C05488=1193.107,194.076,-58.104,-177.783,6.528,148.541
C05489=1193.102,194.324,-58.128,-177.781,6.530,148.540
C05490=1193.099,194.573,-58.150,-177.778,6.532,148.540
C05491=1193.094,194.822,-58.174,-177.775,6.534,148.540
C05492=1193.089,195.071,-58.197,-177.773,6.536,148.539
C05493=1193.085,195.320,-58.221,-177.770,6.537,148.539
C05494=1193.080,195.569,-58.245,-177.767,6.539,148.539
C05495=1193.075,195.818,-58.268,-177.765,6.541,148.538
C05496=1193.071,196.066,-58.292,-177.762,6.543,148.538
C05497=1193.066,196.315,-58.315,-177.760,6.545,148.538
C05498=1193.062,196.564,-58.339,-177.757,6.547,148.537
C05499=1193.057,196.813,-58.363,-177.754,6.548,148.537
C05500=1193.052,197.062,-58.386,-177.752,6.550,148.537
C05501=1193.048,197.311,-58.410,-177.749,6.552,148.536
C05502=1193.043,197.559,-58.434,-177.746,6.554,148.536
C05503=1193.038,197.808,-58.458,-177.743,6.557,148.536
C05504=1193.034,198.057,-58.482,-177.741,6.559,148.536
C05505=1193.029,198.307,-58.505,-177.738,6.560,148.535
C05506=1193.025,198.556,-58.529,-177.736,6.562,148.535
C05507=1193.020,198.804,-58.553,-177.733,6.564,148.535
C05508=1193.016,199.053,-58.576,-177.730,6.566,148.534
C05509=1193.011,199.301,-58.600,-177.728,6.568,148.534
C05510=1193.007,199.550,-58.624,-177.725,6.570,148.534
C05511=1193.002,199.799,-58.648,-177.723,6.572,148.533
C05512=1192.997,200.048,-58.671,-177.720,6.573,148.533
C05513=1192.993,200.296,-58.695,-177.718,6.575,148.533
C05514=1192.988,200.546,-58.719,-177.714,6.578,148.532
C05515=1192.983,200.794,-58.743,-177.712,6.580,148.532
C05516=1192.979,201.044,-58.767,-177.709,6.582,148.532
C05517=1192.975,201.292,-58.791,-177.706,6.583,148.531
C05518=1192.970,201.541,-58.814,-177.704,6.585,148.531
C05519=1192.966,201.790,-58.838,-177.702,6.587,148.531
C05520=1192.960,202.038,-58.863,-177.699,6.589,148.531
C05521=1192.956,202.287,-58.886,-177.696,6.591,148.530
C05522=1192.951,202.536,-58.910,-177.694,6.593,148.530
C05523=1192.947,202.785,-58.934,-177.690,6.595,148.530
C05524=1192.943,203.034,-58.958,-177.688,6.598,148.529
C05525=1192.938,203.283,-58.983,-177.686,6.599,148.529
C05526=1192.933,203.532,-59.006,-177.683,6.601,148.529
C05527=1192.929,203.780,-59.030,-177.680,6.603,148.528
C05528=1192.924,204.029,-59.054,-177.678,6.605,148.528
C05529=1192.920,204.278,-59.078,-177.675,6.607,148.528
C05530=1192.915,204.527,-59.103,-177.673,6.609,148.528
C05531=1192.911,204.775,-59.127,-177.670,6.611,148.527
C05532=1192.906,205.024,-59.151,-177.667,6.613,148.527
C05533=1192.902,205.273,-59.174,-177.664,6.615,148.527
C05534=1192.896,205.522,-59.199,-177.662,6.617,148.526
C05535=1192.893,205.771,-59.223,-177.659,6.619,148.526
C05536=1192.888,206.019,-59.248,-177.657,6.621,148.526
C05537=1192.883,206.268,-59.271,-177.654,6.623,148.525
C05538=1192.878,206.517,-59.296,-177.651,6.625,148.525
C05539=1192.874,206.765,-59.320,-177.648,6.627,148.525
C05540=1192.869,207.015,-59.345,-177.646,6.629,148.524
C05541=1192.865,207.263,-59.369,-177.643,6.631,148.524
C05542=1192.861,207.512,-59.393,-177.641,6.633,148.524
C05543=1192.855,207.761,-59.417,-177.638,6.635,148.524
C05544=1192.851,208.009,-59.441,-177.635,6.636,148.523
C05545=1192.847,208.258,-59.465,-177.632,6.639,148.523
C05546=1192.842,208.507,-59.490,-177.630,6.641,148.523
C05547=1192.838,208.756,-59.514,-177.627,6.643,148.523
C05548=1192.832,209.004,-59.539,-177.625,6.645,148.522
C05549=1192.829,209.253,-59.563,-177.622,6.647,148.522
C05550=1192.824,209.502,-59.587,-177.620,6.649,148.522
C05551=1192.819,209.751,-59.612,-177.617,6.651,148.521
C05552=1192.815,210.000,-59.636,-177.614,6.653,148.521
C05553=1192.810,210.248,-59.661,-177.611,6.655,148.521
C05554=1192.805,210.519,-59.687,-177.609,6.657,148.520
C05555=1192.800,210.789,-59.713,-177.605,6.659,148.520
C05556=1192.796,211.060,-59.740,-177.603,6.661,148.520
C05557=1192.791,211.330,-59.767,-177.600,6.664,148.519
C05558=1192.785,211.579,-59.792,-177.597,6.666,148.519
C05559=1192.781,211.827,-59.816,-177.595,6.668,148.519
C05560=1192.777,212.077,-59.841,-177.592,6.670,148.519
C05561=1192.772,212.325,-59.865,-177.589,6.672,148.518
C05562=1192.767,212.574,-59.889,-177.587,6.675,148.518
C05563=1192.763,212.823,-59.914,-177.584,6.676,148.518
C05564=1192.758,213.072,-59.939,-177.581,6.678,148.518
C05565=1192.754,213.320,-59.963,-177.579,6.680,148.517
C05566=1192.749,213.569,-59.988,-177.577,6.682,148.517
C05567=1192.745,213.817,-60.012,-177.574,6.684,148.517
C05568=1192.741,214.067,-60.037,-177.571,6.687,148.516
C05569=1192.736,214.315,-60.062,-177.568,6.688,148.516
C05570=1192.731,214.564,-60.086,-177.566,6.691,148.516
C05571=1192.727,214.813,-60.111,-177.563,6.692,148.516
C05572=1192.722,215.062,-60.135,-177.561,6.694,148.515
C05573=1192.717,215.310,-60.161,-177.557,6.697,148.515
C05574=1192.713,215.559,-60.185,-177.555,6.699,148.515
C05575=1192.708,215.808,-60.210,-177.553,6.701,148.515
C05576=1192.705,216.057,-60.234,-177.550,6.703,148.514
C05577=1192.700,216.305,-60.260,-177.547,6.704,148.514
C05578=1192.695,216.553,-60.284,-177.545,6.707,148.514
C05579=1192.691,216.803,-60.309,-177.542,6.709,148.514
C05580=1192.686,217.051,-60.333,-177.539,6.711,148.513
C05581=1192.681,217.300,-60.359,-177.537,6.713,148.513
C05582=1192.677,217.549,-60.383,-177.534,6.716,148.513
C05583=1192.672,217.797,-60.408,-177.531,6.718,148.512
C05584=1192.668,218.046,-60.433,-177.529,6.719,148.512
C05585=1192.663,218.294,-60.458,-177.526,6.722,148.512
C05586=1192.659,218.544,-60.483,-177.524,6.723,148.512
C05587=1192.654,218.792,-60.508,-177.521,6.726,148.511
C05588=1192.650,219.041,-60.533,-177.518,6.728,148.511
C05589=1192.645,219.290,-60.557,-177.516,6.730,148.511
C05590=1192.641,219.539,-60.583,-177.513,6.732,148.511
C05591=1192.636,219.787,-60.607,-177.510,6.734,148.510
C05592=1192.632,220.036,-60.633,-177.508,6.737,148.510
C05593=1192.627,220.285,-60.657,-177.505,6.738,148.510
C05594=1192.623,220.533,-60.683,-177.502,6.740,148.510
C05595=1192.618,220.782,-60.707,-177.500,6.742,148.509
C05596=1192.614,221.031,-60.733,-177.497,6.745,148.509
C05597=1192.609,221.279,-60.758,-177.494,6.747,148.509
C05598=1192.605,221.529,-60.783,-177.492,6.749,148.508
C05599=1192.600,221.777,-60.808,-177.490,6.751,148.508
C05600=1192.596,222.025,-60.833,-177.486,6.754,148.508
C05601=1192.591,222.274,-60.858,-177.484,6.755,148.508
C05602=1192.587,222.523,-60.884,-177.482,6.757,148.508
C05603=1192.582,222.772,-60.908,-177.479,6.759,148.507
C05604=1192.578,223.020,-60.934,-177.476,6.762,148.507
C05605=1192.573,223.269,-60.958,-177.473,6.764,148.507
C05606=1192.569,223.518,-60.984,-177.471,6.766,148.507
C05607=1192.564,223.766,-61.009,-177.468,6.768,148.506
C05608=1192.560,224.015,-61.034,-177.465,6.771,148.506
C05609=1192.555,224.263,-61.060,-177.463,6.773,148.506
C05610=1192.550,224.513,-61.085,-177.460,6.774,148.505
C05611=1192.546,224.760,-61.110,-177.458,6.777,148.505
C05612=1192.542,225.009,-61.135,-177.455,6.779,148.505
C05613=1192.537,225.259,-61.160,-177.452,6.781,148.505
C05614=1192.533,225.507,-61.186,-177.450,6.783,148.505
C05615=1192.528,225.756,-61.212,-177.447,6.785,148.504
C05616=1192.523,226.004,-61.236,-177.444,6.788,148.504
C05617=1192.519,226.253,-61.262,-177.442,6.790,148.504
C05618=1192.515,226.502,-61.288,-177.439,6.792,148.504
C05619=1192.510,226.750,-61.313,-177.437,6.793,148.503
C05620=1192.505,226.999,-61.338,-177.434,6.796,148.503
C05621=1192.501,227.248,-61.364,-177.431,6.798,148.503
C05622=1192.496,227.496,-61.389,-177.429,6.800,148.502
C05623=1192.492,227.745,-61.415,-177.426,6.802,148.502
C05624=1192.487,227.994,-61.440,-177.423,6.805,148.502
C05625=1192.483,228.243,-61.465,-177.421,6.807,148.502
C05626=1192.478,228.491,-61.491,-177.418,6.809,148.502
C05627=1192.474,228.740,-61.517,-177.415,6.811,148.501
C05628=1192.469,228.988,-61.542,-177.413,6.814,148.501
C05629=1192.465,229.237,-61.568,-177.410,6.815,148.501
C05630=1192.460,229.486,-61.593,-177.408,6.817,148.501
C05631=1192.456,229.735,-61.618,-177.405,6.820,148.501
C05632=1192.451,229.983,-61.644,-177.402,6.822,148.500
C05633=1192.447,230.232,-61.670,-177.400,6.824,148.500
C05634=1192.443,230.480,-61.695,-177.397,6.827,148.500
C05635=1192.438,230.729,-61.721,-177.394,6.829,148.499
C05636=1192.434,230.977,-61.747,-177.392,6.831,148.499
C05637=1192.429,231.226,-61.772,-177.390,6.833,148.499
C05638=1192.424,231.474,-61.798,-177.387,6.836,148.499
C05639=1192.420,231.723,-61.823,-177.384,6.838,148.499
C05640=1192.416,231.972,-61.849,-177.382,6.839,148.498
C05641=1192.412,232.221,-61.875,-177.379,6.842,148.498
C05642=1192.407,232.469,-61.900,-177.376,6.844,148.498
C05643=1192.402,232.718,-61.927,-177.374,6.846,148.498
C05644=1192.398,232.967,-61.952,-177.371,6.848,148.498
C05645=1192.393,233.215,-61.978,-177.369,6.851,148.497
C05646=1192.389,233.464,-62.004,-177.366,6.853,148.497
C05647=1192.385,233.712,-62.029,-177.363,6.855,148.497
C05648=1192.380,233.961,-62.055,-177.361,6.858,148.497
C05649=1192.375,234.210,-62.081,-177.358,6.860,148.496
C05650=1192.370,234.458,-62.107,-177.356,6.862,148.496
C05651=1192.366,234.707,-62.132,-177.353,6.864,148.496
C05652=1192.362,234.956,-62.158,-177.350,6.867,148.496
C05653=1192.358,235.204,-62.184,-177.348,6.868,148.496
C05654=1192.353,235.453,-62.211,-177.345,6.871,148.495
C05655=1192.348,235.701,-62.236,-177.342,6.873,148.495
C05656=1192.344,235.950,-62.262,-177.340,6.875,148.495
C05657=1192.339,236.198,-62.288,-177.337,6.878,148.495
C05658=1192.335,236.470,-62.316,-177.334,6.880,148.494
C05659=1192.329,236.742,-62.345,-177.331,6.883,148.494
C05660=1192.325,237.013,-62.374,-177.329,6.885,148.494
C05661=1192.320,237.284,-62.401,-177.326,6.887,148.494
C05662=1192.316,237.533,-62.427,-177.323,6.889,148.493
C05663=1192.311,237.782,-62.453,-177.321,6.892,148.493
C05664=1192.307,238.030,-62.480,-177.318,6.894,148.493
C05665=1192.302,238.279,-62.506,-177.316,6.896,148.493
C05666=1192.297,238.528,-62.532,-177.313,6.899,148.493
C05667=1192.293,238.776,-62.558,-177.310,6.901,148.493
C05668=1192.289,239.025,-62.584,-177.308,6.903,148.492
C05669=1192.284,239.274,-62.610,-177.305,6.906,148.492
C05670=1192.280,239.522,-62.637,-177.302,6.908,148.492
C05671=1192.276,239.771,-62.662,-177.300,6.911,148.492
C05672=1192.271,240.020,-62.689,-177.297,6.912,148.492
C05673=1192.266,240.267,-62.715,-177.295,6.915,148.491
C05674=1192.262,240.516,-62.741,-177.292,6.917,148.491
C05675=1192.257,240.765,-62.767,-177.289,6.919,148.491
C05676=1192.253,241.013,-62.793,-177.287,6.921,148.491
C05677=1192.249,241.262,-62.819,-177.284,6.924,148.491
C05678=1192.244,241.511,-62.846,-177.281,6.926,148.490
C05679=1192.240,241.760,-62.872,-177.279,6.928,148.490
C05680=1192.235,242.008,-62.899,-177.276,6.931,148.490
C05681=1192.230,242.256,-62.924,-177.274,6.933,148.490
C05682=1192.226,242.505,-62.952,-177.271,6.935,148.490
C05683=1192.222,242.753,-62.977,-177.269,6.938,148.489
C05684=1192.218,243.002,-63.004,-177.266,6.940,148.489
C05685=1192.213,243.251,-63.030,-177.263,6.943,148.489
C05686=1192.209,243.499,-63.057,-177.261,6.944,148.489
C05687=1192.204,243.748,-63.083,-177.258,6.947,148.489
C05688=1192.200,243.996,-63.109,-177.255,6.949,148.488
C05689=1192.195,244.245,-63.136,-177.253,6.951,148.488
C05690=1192.191,244.494,-63.162,-177.250,6.953,148.488
C05691=1192.186,244.742,-63.189,-177.248,6.956,148.488
C05692=1192.182,244.991,-63.215,-177.245,6.958,148.488
C05693=1192.177,245.239,-63.242,-177.242,6.961,148.488
C05694=1192.173,245.488,-63.268,-177.240,6.963,148.487
C05695=1192.169,245.737,-63.295,-177.238,6.965,148.487
C05696=1192.165,245.985,-63.321,-177.235,6.968,148.487
C05697=1192.159,246.233,-63.347,-177.232,6.970,148.487
C05698=1192.154,246.482,-63.374,-177.229,6.973,148.487
C05699=1192.151,246.730,-63.401,-177.227,6.975,148.486
C05700=1192.146,246.979,-63.427,-177.225,6.977,148.486
C05701=1192.142,247.227,-63.454,-177.221,6.980,148.486
C05702=1192.137,247.476,-63.481,-177.219,6.982,148.486
C05703=1192.133,247.724,-63.507,-177.217,6.985,148.486
C05704=1192.128,247.973,-63.534,-177.214,6.987,148.486
C05705=1192.123,248.222,-63.561,-177.212,6.989,148.485
C05706=1192.120,248.470,-63.587,-177.209,6.991,148.485
C05707=1192.116,248.719,-63.615,-177.206,6.994,148.485
C05708=1192.111,248.968,-63.641,-177.203,6.996,148.485
C05709=1192.107,249.216,-63.667,-177.201,6.998,148.485
C05710=1192.102,249.465,-63.694,-177.198,7.001,148.485
C05711=1192.097,249.713,-63.721,-177.196,7.003,148.484
C05712=1192.093,249.961,-63.748,-177.194,7.005,148.484
C05713=1192.089,250.210,-63.775,-177.190,7.008,148.484
C05714=1192.084,250.459,-63.801,-177.188,7.010,148.484
C05715=1192.080,250.707,-63.828,-177.185,7.013,148.484
C05716=1192.075,250.956,-63.855,-177.183,7.015,148.484
C05717=1192.071,251.204,-63.882,-177.181,7.017,148.483
C05718=1192.067,251.452,-63.908,-177.177,7.020,148.483
C05719=1192.062,251.701,-63.935,-177.175,7.022,148.483
C05720=1192.057,251.949,-63.962,-177.172,7.025,148.483
C05721=1192.053,252.198,-63.990,-177.170,7.027,148.483
C05722=1192.049,252.446,-64.016,-177.167,7.030,148.483
C05723=1192.045,252.695,-64.043,-177.165,7.032,148.482
C05724=1192.040,252.944,-64.071,-177.162,7.035,148.482
C05725=1192.035,253.192,-64.098,-177.159,7.036,148.482
C05726=1192.031,253.440,-64.124,-177.157,7.039,148.482
C05727=1192.027,253.689,-64.151,-177.154,7.042,148.482
C05728=1192.022,253.937,-64.178,-177.152,7.043,148.482
C05729=1192.017,254.186,-64.205,-177.149,7.046,148.481
C05730=1192.013,254.434,-64.232,-177.147,7.049,148.481
C05731=1192.009,254.683,-64.259,-177.144,7.051,148.481
C05732=1192.005,254.932,-64.286,-177.141,7.053,148.481
C05733=1192.000,255.180,-64.313,-177.138,7.056,148.481
C05734=1191.996,255.429,-64.340,-177.136,7.058,148.481
C05735=1191.991,255.677,-64.367,-177.133,7.061,148.481
C05736=1191.987,255.925,-64.395,-177.131,7.063,148.480
C05737=1191.982,256.174,-64.423,-177.129,7.065,148.480
C05738=1191.979,256.423,-64.449,-177.126,7.068,148.480
C05739=1191.974,256.671,-64.476,-177.123,7.070,148.480
C05740=1191.969,256.920,-64.503,-177.121,7.073,148.480
C05741=1191.965,257.168,-64.530,-177.118,7.075,148.480
C05742=1191.960,257.416,-64.558,-177.115,7.078,148.479
C05743=1191.956,257.665,-64.585,-177.113,7.080,148.479
C05744=1191.952,257.914,-64.612,-177.110,7.083,148.479
C05745=1191.947,258.162,-64.640,-177.108,7.085,148.479
C05746=1191.943,258.410,-64.667,-177.105,7.088,148.479
C05747=1191.938,258.658,-64.694,-177.103,7.090,148.479
C05748=1191.934,258.908,-64.722,-177.100,7.093,148.479
C05749=1191.929,259.156,-64.749,-177.097,7.095,148.478
C05750=1191.925,259.404,-64.777,-177.095,7.098,148.478
C05751=1191.920,259.652,-64.804,-177.092,7.100,148.478
C05752=1191.916,259.902,-64.831,-177.089,7.103,148.478
C05753=1191.912,260.150,-64.859,-177.087,7.105,148.478
C05754=1191.907,260.398,-64.886,-177.084,7.108,148.478
C05755=1191.902,260.647,-64.913,-177.082,7.110,148.478
C05756=1191.899,260.895,-64.941,-177.079,7.113,148.478
C05757=1191.894,261.144,-64.968,-177.076,7.115,148.477
C05758=1191.890,261.392,-64.996,-177.074,7.118,148.477
C05759=1191.885,261.640,-65.023,-177.072,7.120,148.477
C05760=1191.881,261.889,-65.051,-177.068,7.122,148.477
C05761=1191.877,262.137,-65.078,-177.066,7.125,148.477
C05762=1191.871,262.410,-65.109,-177.064,7.128,148.477
C05763=1191.867,262.683,-65.139,-177.060,7.130,148.476
C05764=1191.862,262.955,-65.169,-177.058,7.133,148.476
C05765=1191.857,263.229,-65.200,-177.055,7.136,148.476
C05766=1191.853,263.477,-65.227,-177.052,7.138,148.476
C05767=1191.848,263.725,-65.255,-177.050,7.141,148.476
C05768=1191.844,263.974,-65.282,-177.047,7.143,148.476
C05769=1191.840,264.222,-65.310,-177.044,7.146,148.476
C05770=1191.835,264.471,-65.337,-177.042,7.148,148.476
C05771=1191.832,264.719,-65.365,-177.039,7.151,148.476
C05772=1191.827,264.967,-65.393,-177.037,7.153,148.475
C05773=1191.822,265.216,-65.420,-177.034,7.156,148.475
C05774=1191.818,265.464,-65.448,-177.032,7.158,148.475
C05775=1191.813,265.713,-65.476,-177.029,7.161,148.475
C05776=1191.809,265.961,-65.503,-177.027,7.163,148.475
C05777=1191.805,266.209,-65.531,-177.024,7.166,148.475
C05778=1191.800,266.458,-65.559,-177.022,7.168,148.475
C05779=1191.796,266.706,-65.587,-177.019,7.171,148.475
C05780=1191.792,266.955,-65.615,-177.016,7.173,148.474
C05781=1191.787,267.203,-65.642,-177.014,7.176,148.474
C05782=1191.783,267.452,-65.671,-177.011,7.179,148.474
C05783=1191.778,267.700,-65.699,-177.009,7.181,148.474
C05784=1191.774,267.948,-65.726,-177.006,7.184,148.474
C05785=1191.770,268.197,-65.754,-177.003,7.186,148.474
C05786=1191.765,268.445,-65.782,-177.001,7.189,148.474
C05787=1191.761,268.694,-65.810,-176.998,7.191,148.474
C05788=1191.757,268.942,-65.837,-176.996,7.194,148.474
C05789=1191.753,269.191,-65.866,-176.993,7.196,148.473
C05790=1191.748,269.439,-65.894,-176.990,7.199,148.473
C05791=1191.743,269.687,-65.922,-176.988,7.202,148.473
C05792=1191.740,269.935,-65.950,-176.986,7.204,148.473
C05793=1191.734,270.184,-65.977,-176.982,7.207,148.473
C05794=1191.730,270.433,-66.006,-176.980,7.209,148.473
C05795=1191.726,270.681,-66.033,-176.977,7.212,148.473
C05796=1191.722,270.930,-66.062,-176.975,7.214,148.473
C05797=1191.717,271.177,-66.090,-176.973,7.217,148.473
C05798=1191.713,271.426,-66.118,-176.969,7.220,148.472
C05799=1191.708,271.674,-66.146,-176.967,7.222,148.472
C05800=1191.704,271.922,-66.174,-176.965,7.225,148.472
C05801=1191.700,272.171,-66.203,-176.962,7.227,148.472
C05802=1191.695,272.419,-66.231,-176.959,7.230,148.472
C05803=1191.691,272.667,-66.259,-176.957,7.232,148.472
C05804=1191.686,272.916,-66.287,-176.954,7.235,148.472
C05805=1191.682,273.165,-66.315,-176.952,7.238,148.472
C05806=1191.677,273.413,-66.343,-176.949,7.240,148.472
C05807=1191.673,273.662,-66.371,-176.947,7.243,148.472
C05808=1191.669,273.910,-66.401,-176.944,7.245,148.471
C05809=1191.665,274.158,-66.428,-176.941,7.248,148.471
C05810=1191.661,274.406,-66.457,-176.939,7.251,148.471
C05811=1191.656,274.654,-66.485,-176.937,7.253,148.471
C05812=1191.652,274.903,-66.513,-176.934,7.256,148.471
C05813=1191.647,275.151,-66.541,-176.931,7.258,148.471
C05814=1191.644,275.400,-66.570,-176.929,7.261,148.471
C05815=1191.638,275.648,-66.598,-176.926,7.263,148.471
C05816=1191.635,275.897,-66.626,-176.924,7.266,148.471
C05817=1191.630,276.145,-66.654,-176.921,7.269,148.471
C05818=1191.626,276.393,-66.683,-176.919,7.271,148.471
C05819=1191.622,276.642,-66.712,-176.916,7.274,148.470
C05820=1191.617,276.890,-66.740,-176.913,7.277,148.470
C05821=1191.613,277.138,-66.769,-176.911,7.279,148.470
C05822=1191.608,277.386,-66.796,-176.908,7.282,148.470
C05823=1191.604,277.635,-66.825,-176.906,7.284,148.470
C05824=1191.600,277.883,-66.855,-176.903,7.287,148.470
C05825=1191.595,278.131,-66.882,-176.900,7.290,148.470
C05826=1191.591,278.380,-66.911,-176.898,7.292,148.470
C05827=1191.587,278.628,-66.939,-176.895,7.295,148.470
C05828=1191.582,278.876,-66.968,-176.893,7.297,148.470
C05829=1191.578,279.125,-66.997,-176.890,7.300,148.470
C05830=1191.574,279.373,-67.025,-176.888,7.303,148.470
C05831=1191.569,279.622,-67.054,-176.885,7.306,148.469
C05832=1191.566,279.870,-67.082,-176.883,7.309,148.469
C05833=1191.561,280.118,-67.111,-176.879,7.311,148.469
C05834=1191.556,280.366,-67.140,-176.877,7.313,148.469
C05835=1191.552,280.614,-67.168,-176.875,7.316,148.469
C05836=1191.548,280.863,-67.197,-176.872,7.319,148.469
C05837=1191.543,281.111,-67.226,-176.870,7.322,148.469
C05838=1191.539,281.359,-67.254,-176.867,7.325,148.469
C05839=1191.535,281.608,-67.283,-176.865,7.327,148.469
C05840=1191.530,281.856,-67.312,-176.862,7.330,148.469
C05841=1191.525,282.105,-67.341,-176.859,7.333,148.469
C05842=1191.522,282.353,-67.369,-176.857,7.335,148.468
C05843=1191.517,282.601,-67.398,-176.854,7.338,148.468
C05844=1191.513,282.850,-67.428,-176.851,7.341,148.468
C05845=1191.509,283.098,-67.455,-176.849,7.343,148.468
C05846=1191.505,283.346,-67.485,-176.847,7.346,148.468
C05847=1191.500,283.595,-67.514,-176.844,7.349,148.468
C05848=1191.495,283.842,-67.543,-176.842,7.351,148.468
C05849=1191.491,284.091,-67.571,-176.839,7.354,148.468
C05850=1191.487,284.339,-67.600,-176.837,7.356,148.468
C05851=1191.483,284.588,-67.629,-176.834,7.359,148.468
C05852=1191.478,284.836,-67.658,-176.831,7.362,148.468
C05853=1191.474,285.085,-67.687,-176.829,7.364,148.468
C05854=1191.469,285.333,-67.716,-176.826,7.367,148.468
C05855=1191.465,285.580,-67.745,-176.823,7.370,148.468
C05856=1191.461,285.829,-67.773,-176.821,7.372,148.468
C05857=1191.457,286.077,-67.803,-176.818,7.375,148.468
C05858=1191.453,286.325,-67.832,-176.816,7.378,148.468
C05859=1191.448,286.574,-67.861,-176.814,7.380,148.467
C05860=1191.443,286.822,-67.890,-176.811,7.383,148.467
C05861=1191.440,287.070,-67.919,-176.808,7.386,148.467
C05862=1191.435,287.319,-67.948,-176.806,7.388,148.467
C05863=1191.431,287.567,-67.977,-176.803,7.391,148.467
C05864=1191.426,287.815,-68.006,-176.801,7.394,148.467
C05865=1191.422,288.064,-68.035,-176.798,7.397,148.467
C05866=1191.418,288.338,-68.068,-176.795,7.400,148.467
C05867=1191.412,288.613,-68.100,-176.792,7.403,148.467
C05868=1191.408,288.886,-68.132,-176.789,7.406,148.467
C05869=1191.403,289.162,-68.165,-176.787,7.409,148.467
C05870=1191.398,289.409,-68.194,-176.784,7.411,148.467
C05871=1191.394,289.658,-68.224,-176.782,7.414,148.467
C05872=1191.390,289.906,-68.252,-176.779,7.417,148.467
C05873=1191.386,290.154,-68.281,-176.777,7.420,148.467
C05874=1191.382,290.403,-68.311,-176.774,7.423,148.467
C05875=1191.378,290.651,-68.340,-176.771,7.426,148.467
C05876=1191.374,290.899,-68.370,-176.769,7.429,148.467
C05877=1191.369,291.147,-68.399,-176.767,7.431,148.467
C05878=1191.365,291.395,-68.428,-176.764,7.434,148.467
C05879=1191.360,291.643,-68.458,-176.761,7.437,148.467
C05880=1191.356,291.892,-68.486,-176.759,7.439,148.466
C05881=1191.351,292.141,-68.516,-176.756,7.442,148.466
C05882=1191.347,292.389,-68.546,-176.754,7.445,148.466
C05883=1191.343,292.637,-68.575,-176.751,7.447,148.466
C05884=1191.339,292.886,-68.605,-176.749,7.450,148.466
C05885=1191.334,293.133,-68.634,-176.746,7.453,148.466
C05886=1191.330,293.381,-68.663,-176.743,7.456,148.466
C05887=1191.325,293.630,-68.693,-176.741,7.458,148.466
C05888=1191.321,293.878,-68.722,-176.738,7.461,148.466
C05889=1191.317,294.126,-68.752,-176.736,7.464,148.466
C05890=1191.313,294.374,-68.782,-176.734,7.466,148.466
C05891=1191.309,294.622,-68.811,-176.731,7.469,148.466
C05892=1191.305,294.870,-68.841,-176.728,7.472,148.466
C05893=1191.300,295.119,-68.871,-176.725,7.475,148.466
C05894=1191.296,295.367,-68.900,-176.723,7.478,148.466
C05895=1191.291,295.616,-68.930,-176.721,7.481,148.466
C05896=1191.287,295.864,-68.959,-176.718,7.484,148.466
C05897=1191.283,296.112,-68.988,-176.716,7.486,148.466
C05898=1191.279,296.360,-69.018,-176.713,7.489,148.466
C05899=1191.275,296.608,-69.048,-176.710,7.492,148.466
C05900=1191.270,296.857,-69.078,-176.708,7.495,148.466
C05901=1191.266,297.105,-69.108,-176.706,7.497,148.466
C05902=1191.262,297.353,-69.137,-176.703,7.500,148.466
C05903=1191.258,297.601,-69.167,-176.701,7.503,148.466
C05904=1191.253,297.849,-69.197,-176.698,7.506,148.466
C05905=1191.249,298.098,-69.227,-176.696,7.509,148.466
C05906=1191.245,298.346,-69.256,-176.693,7.512,148.466
C05907=1191.240,298.594,-69.286,-176.690,7.515,148.466
C05908=1191.236,298.842,-69.316,-176.688,7.517,148.466
C05909=1191.232,299.090,-69.346,-176.685,7.520,148.466
C05910=1191.227,299.339,-69.375,-176.683,7.523,148.466
C05911=1191.224,299.586,-69.405,-176.680,7.526,148.466
C05912=1191.219,299.835,-69.436,-176.678,7.528,148.466
C05913=1191.214,300.083,-69.465,-176.676,7.531,148.466
C05914=1191.211,300.331,-69.495,-176.673,7.534,148.466
C05915=1191.206,300.579,-69.525,-176.670,7.537,148.466
C05916=1191.202,300.828,-69.555,-176.668,7.539,148.466
C05917=1191.198,301.075,-69.585,-176.665,7.542,148.466
C05918=1191.193,301.324,-69.615,-176.663,7.545,148.466
C05919=1191.189,301.571,-69.645,-176.660,7.548,148.466
C05920=1191.185,301.820,-69.675,-176.658,7.551,148.466
C05921=1191.180,302.068,-69.705,-176.655,7.554,148.466
C05922=1191.176,302.316,-69.735,-176.652,7.557,148.465
C05923=1191.172,302.564,-69.765,-176.650,7.560,148.466
C05924=1191.168,302.813,-69.795,-176.648,7.562,148.466
C05925=1191.164,303.061,-69.825,-176.645,7.565,148.466
C05926=1191.159,303.309,-69.856,-176.643,7.568,148.466
C05927=1191.155,303.557,-69.886,-176.640,7.571,148.466
C05928=1191.150,303.805,-69.916,-176.638,7.573,148.465
C05929=1191.146,304.053,-69.946,-176.635,7.576,148.465
C05930=1191.142,304.301,-69.975,-176.633,7.580,148.466
C05931=1191.137,304.549,-70.006,-176.630,7.583,148.466
C05932=1191.133,304.797,-70.036,-176.628,7.585,148.466
C05933=1191.129,305.046,-70.067,-176.625,7.588,148.466
C05934=1191.125,305.294,-70.097,-176.622,7.591,148.466
C05935=1191.120,305.542,-70.127,-176.620,7.594,148.466
C05936=1191.117,305.790,-70.157,-176.618,7.596,148.465
C05937=1191.112,306.038,-70.188,-176.615,7.599,148.466
C05938=1191.108,306.286,-70.217,-176.613,7.602,148.466
C05939=1191.103,306.534,-70.248,-176.610,7.605,148.466
C05940=1191.100,306.783,-70.279,-176.607,7.608,148.466
C05941=1191.095,307.031,-70.309,-176.605,7.611,148.466
C05942=1191.091,307.279,-70.339,-176.603,7.614,148.466
C05943=1191.086,307.527,-70.370,-176.600,7.617,148.466
C05944=1191.082,307.775,-70.400,-176.597,7.620,148.466
C05945=1191.078,308.023,-70.430,-176.595,7.622,148.466
C05946=1191.074,308.272,-70.461,-176.593,7.625,148.466
C05947=1191.070,308.519,-70.491,-176.590,7.628,148.466
C05948=1191.065,308.767,-70.522,-176.588,7.631,148.466
C05949=1191.061,309.015,-70.551,-176.585,7.634,148.466
C05950=1191.057,309.264,-70.582,-176.583,7.637,148.466
C05951=1191.052,309.512,-70.613,-176.580,7.640,148.466
C05952=1191.048,309.760,-70.643,-176.578,7.643,148.466
C05953=1191.044,310.008,-70.674,-176.575,7.646,148.466
C05954=1191.039,310.256,-70.705,-176.573,7.648,148.466
C05955=1191.036,310.504,-70.735,-176.570,7.651,148.466
C05956=1191.031,310.753,-70.765,-176.568,7.654,148.466
C05957=1191.026,311.001,-70.796,-176.565,7.658,148.466
C05958=1191.023,311.248,-70.826,-176.563,7.661,148.466
C05959=1191.019,311.497,-70.858,-176.561,7.663,148.466
C05960=1191.014,311.745,-70.888,-176.558,7.666,148.466
C05961=1191.010,311.992,-70.918,-176.556,7.669,148.466
C05962=1191.006,312.241,-70.950,-176.553,7.672,148.466
C05963=1191.001,312.489,-70.980,-176.550,7.675,148.466
C05964=1190.998,312.737,-71.011,-176.548,7.677,148.466
C05965=1190.993,312.985,-71.041,-176.546,7.681,148.466
C05966=1190.989,313.233,-71.072,-176.543,7.684,148.466
C05967=1190.984,313.481,-71.103,-176.540,7.687,148.466
C05968=1190.980,313.729,-71.133,-176.538,7.690,148.467
C05969=1190.976,313.978,-71.165,-176.536,7.692,148.466
C05970=1190.972,314.253,-71.199,-176.533,7.696,148.466
C05971=1190.967,314.530,-71.234,-176.530,7.699,148.466
C05972=1190.962,314.807,-71.268,-176.527,7.702,148.466
C05973=1190.957,315.083,-71.302,-176.525,7.705,148.467
C05974=1190.953,315.331,-71.333,-176.522,7.708,148.467
C05975=1190.948,315.579,-71.364,-176.520,7.711,148.467
C05976=1190.945,315.827,-71.394,-176.517,7.715,148.467
C05977=1190.940,316.075,-71.425,-176.515,7.717,148.467
C05978=1190.937,316.323,-71.457,-176.513,7.720,148.467
C05979=1190.932,316.571,-71.488,-176.510,7.723,148.467
C05980=1190.927,316.819,-71.518,-176.508,7.726,148.467
C05981=1190.923,317.068,-71.550,-176.505,7.729,148.467
C05982=1190.920,317.315,-71.580,-176.503,7.732,148.467
C05983=1190.915,317.563,-71.611,-176.501,7.735,148.467
C05984=1190.911,317.812,-71.642,-176.498,7.738,148.467
C05985=1190.907,318.060,-71.673,-176.496,7.741,148.467
C05986=1190.903,318.308,-71.705,-176.493,7.744,148.467
C05987=1190.898,318.556,-71.736,-176.490,7.747,148.467
C05988=1190.894,318.804,-71.766,-176.489,7.749,148.467
C05989=1190.890,319.052,-71.798,-176.486,7.753,148.467
C05990=1190.885,319.300,-71.829,-176.483,7.756,148.467
C05991=1190.881,319.548,-71.860,-176.481,7.759,148.468
C05992=1190.877,319.795,-71.892,-176.478,7.762,148.468
C05993=1190.874,320.044,-71.922,-176.476,7.765,148.468
C05994=1190.869,320.292,-71.953,-176.474,7.767,148.468
C05995=1190.865,320.540,-71.985,-176.471,7.770,148.468
C05996=1190.861,320.788,-72.016,-176.469,7.774,148.468
C05997=1190.857,321.035,-72.047,-176.466,7.777,148.468
C05998=1190.853,321.284,-72.078,-176.464,7.780,148.468
C05999=1190.848,321.531,-72.110,-176.462,7.782,148.468
C06000=1190.844,321.780,-72.141,-176.459,7.785,148.468
C06001=1190.840,322.027,-72.172,-176.457,7.789,148.468
C06002=1190.836,322.276,-72.203,-176.454,7.792,148.468
C06003=1190.832,322.523,-72.235,-176.452,7.795,148.469
C06004=1190.828,322.772,-72.266,-176.449,7.798,148.469
C06005=1190.823,323.019,-72.298,-176.447,7.800,148.469
C06006=1190.818,323.268,-72.329,-176.445,7.803,148.469
C06007=1190.814,323.515,-72.361,-176.442,7.806,148.469
C06008=1190.810,323.764,-72.392,-176.440,7.810,148.469
C06009=1190.806,324.011,-72.423,-176.437,7.813,148.469
C06010=1190.802,324.260,-72.454,-176.435,7.816,148.469
C06011=1190.798,324.507,-72.486,-176.433,7.818,148.469
C06012=1190.794,324.755,-72.518,-176.430,7.822,148.469
C06013=1190.790,325.004,-72.549,-176.428,7.825,148.469
C06014=1190.786,325.251,-72.580,-176.426,7.828,148.469
C06015=1190.782,325.500,-72.612,-176.423,7.831,148.469
C06016=1190.776,325.748,-72.644,-176.421,7.834,148.470
C06017=1190.773,325.996,-72.675,-176.418,7.836,148.470
C06018=1190.768,326.243,-72.707,-176.416,7.840,148.470
C06019=1190.764,326.492,-72.738,-176.414,7.843,148.470
C06020=1190.760,326.739,-72.770,-176.411,7.846,148.470
C06021=1190.756,326.987,-72.801,-176.409,7.849,148.470
C06022=1190.752,327.236,-72.834,-176.406,7.852,148.470
C06023=1190.747,327.483,-72.865,-176.404,7.855,148.470
C06024=1190.744,327.732,-72.896,-176.402,7.858,148.470
C06025=1190.739,327.979,-72.928,-176.399,7.861,148.470
C06026=1190.736,328.227,-72.960,-176.397,7.864,148.471
C06027=1190.731,328.475,-72.992,-176.394,7.867,148.471
C06028=1190.727,328.723,-73.023,-176.392,7.871,148.471
C06029=1190.723,328.971,-73.055,-176.390,7.873,148.471
C06030=1190.719,329.219,-73.086,-176.388,7.876,148.471
C06031=1190.714,329.467,-73.119,-176.385,7.879,148.471
C06032=1190.710,329.715,-73.151,-176.383,7.882,148.471
C06033=1190.706,329.962,-73.182,-176.380,7.886,148.471
C06034=1190.702,330.211,-73.214,-176.378,7.889,148.471
C06035=1190.697,330.458,-73.246,-176.376,7.892,148.472
C06036=1190.693,330.707,-73.277,-176.374,7.895,148.472
C06037=1190.689,330.955,-73.310,-176.371,7.898,148.472
C06038=1190.685,331.202,-73.341,-176.369,7.901,148.472
C06039=1190.681,331.450,-73.373,-176.366,7.904,148.472
C06040=1190.676,331.699,-73.405,-176.364,7.907,148.472
C06041=1190.672,331.946,-73.437,-176.362,7.911,148.472
C06042=1190.668,332.194,-73.469,-176.360,7.913,148.472
C06043=1190.664,332.442,-73.501,-176.357,7.916,148.473
C06044=1190.660,332.690,-73.533,-176.355,7.919,148.473
C06045=1190.656,332.938,-73.564,-176.352,7.922,148.473
C06046=1190.652,333.186,-73.597,-176.350,7.926,148.473
C06047=1190.648,333.434,-73.629,-176.347,7.929,148.473
C06048=1190.643,333.681,-73.661,-176.345,7.932,148.473
C06049=1190.639,333.929,-73.693,-176.344,7.935,148.473
C06050=1190.636,334.177,-73.725,-176.341,7.938,148.473
C06051=1190.631,334.425,-73.757,-176.339,7.941,148.474
C06052=1190.627,334.673,-73.789,-176.336,7.944,148.474
C06053=1190.622,334.921,-73.822,-176.334,7.948,148.474
C06054=1190.619,335.169,-73.853,-176.331,7.951,148.474
C06055=1190.614,335.417,-73.885,-176.329,7.954,148.474
C06056=1190.610,335.664,-73.918,-176.327,7.956,148.474
C06057=1190.607,335.913,-73.950,-176.325,7.959,148.474
C06058=1190.602,336.161,-73.982,-176.323,7.963,148.475
C06059=1190.598,336.408,-74.014,-176.320,7.966,148.475
C06060=1190.594,336.656,-74.047,-176.318,7.969,148.475
C06061=1190.590,336.904,-74.079,-176.315,7.972,148.475
C06062=1190.586,337.152,-74.111,-176.313,7.976,148.475
C06063=1190.581,337.400,-74.143,-176.311,7.978,148.476
C06064=1190.577,337.647,-74.176,-176.309,7.982,148.476
C06065=1190.573,337.896,-74.208,-176.306,7.985,148.476
C06066=1190.569,338.144,-74.240,-176.304,7.988,148.476
C06067=1190.564,338.391,-74.272,-176.302,7.991,148.476
C06068=1190.561,338.639,-74.305,-176.300,7.995,148.476
C06069=1190.556,338.887,-74.337,-176.298,7.998,148.477
C06070=1190.553,339.135,-74.370,-176.295,8.000,148.477
C06071=1190.548,339.383,-74.402,-176.293,8.003,148.477
C06072=1190.544,339.631,-74.435,-176.291,8.007,148.477
C06073=1190.540,339.878,-74.467,-176.289,8.010,148.477
C06074=1190.535,340.157,-74.503,-176.286,8.013,148.477
C06075=1190.531,340.436,-74.539,-176.283,8.017,148.477
C06076=1190.525,340.715,-74.576,-176.281,8.021,148.478
C06077=1190.521,340.993,-74.613,-176.279,8.024,148.478
C06078=1190.517,341.241,-74.645,-176.276,8.027,148.478
C06079=1190.513,341.489,-74.678,-176.274,8.031,148.478
C06080=1190.509,341.737,-74.710,-176.272,8.034,148.479
C06081=1190.505,341.985,-74.743,-176.270,8.037,148.479
C06082=1190.500,342.232,-74.775,-176.267,8.040,148.479
C06083=1190.496,342.480,-74.808,-176.265,8.044,148.479
C06084=1190.492,342.728,-74.841,-176.263,8.046,148.479
C06085=1190.488,342.976,-74.873,-176.261,8.049,148.479
C06086=1190.484,343.224,-74.906,-176.259,8.053,148.480
C06087=1190.480,343.472,-74.939,-176.256,8.056,148.480
C06088=1190.476,343.719,-74.971,-176.254,8.059,148.480
C06089=1190.472,343.968,-75.004,-176.252,8.063,148.480
C06090=1190.467,344.215,-75.037,-176.250,8.066,148.481
C06091=1190.463,344.462,-75.070,-176.247,8.069,148.481
C06092=1190.458,344.711,-75.102,-176.246,8.072,148.481
C06093=1190.455,344.958,-75.135,-176.243,8.075,148.481
C06094=1190.451,345.207,-75.167,-176.241,8.078,148.481
C06095=1190.446,345.454,-75.200,-176.239,8.082,148.482
C06096=1190.442,345.702,-75.234,-176.237,8.085,148.482
C06097=1190.439,345.949,-75.266,-176.234,8.088,148.482
C06098=1190.435,346.198,-75.299,-176.232,8.092,148.482
C06099=1190.430,346.446,-75.332,-176.231,8.094,148.482
C06100=1190.426,346.693,-75.365,-176.228,8.098,148.483
C06101=1190.422,346.942,-75.397,-176.226,8.101,148.483
C06102=1190.418,347.189,-75.430,-176.224,8.104,148.483
C06103=1190.414,347.437,-75.463,-176.222,8.108,148.483
C06104=1190.410,347.685,-75.496,-176.219,8.111,148.483
C06105=1190.406,347.932,-75.529,-176.217,8.114,148.484
C06106=1190.401,348.180,-75.561,-176.215,8.118,148.484
C06107=1190.397,348.428,-75.595,-176.213,8.120,148.484
C06108=1190.393,348.675,-75.628,-176.211,8.123,148.484
C06109=1190.389,348.923,-75.661,-176.209,8.127,148.485
C06110=1190.384,349.171,-75.694,-176.207,8.130,148.485
C06111=1190.380,349.419,-75.727,-176.205,8.134,148.485
C06112=1190.377,349.666,-75.760,-176.202,8.137,148.485
C06113=1190.372,349.914,-75.792,-176.200,8.140,148.486
C06114=1190.368,350.162,-75.825,-176.198,8.144,148.486
C06115=1190.364,350.410,-75.858,-176.196,8.146,148.486
C06116=1190.360,350.657,-75.892,-176.194,8.149,148.486
C06117=1190.356,350.906,-75.925,-176.192,8.153,148.487
C06118=1190.352,351.154,-75.958,-176.190,8.156,148.487
C06119=1190.348,351.401,-75.991,-176.188,8.160,148.487
C06120=1190.344,351.649,-76.025,-176.185,8.163,148.487
C06121=1190.340,351.897,-76.058,-176.183,8.166,148.488
C06122=1190.336,352.145,-76.091,-176.182,8.169,148.488
C06123=1190.332,352.392,-76.124,-176.180,8.172,148.488
C06124=1190.327,352.640,-76.157,-176.177,8.176,148.488
C06125=1190.323,352.888,-76.190,-176.175,8.179,148.489
C06126=1190.319,353.135,-76.224,-176.173,8.183,148.489
C06127=1190.315,353.383,-76.257,-176.171,8.186,148.489
C06128=1190.311,353.631,-76.290,-176.169,8.189,148.490
C06129=1190.307,353.878,-76.324,-176.167,8.193,148.490
C06130=1190.303,354.126,-76.357,-176.165,8.196,148.490
C06131=1190.299,354.373,-76.390,-176.163,8.199,148.490
C06132=1190.295,354.622,-76.424,-176.161,8.202,148.491
C06133=1190.290,354.870,-76.457,-176.159,8.206,148.491
C06134=1190.286,355.118,-76.490,-176.157,8.209,148.491
C06135=1190.282,355.365,-76.524,-176.155,8.212,148.491
C06136=1190.278,355.613,-76.558,-176.153,8.216,148.492
C06137=1190.274,355.860,-76.591,-176.151,8.219,148.492
C06138=1190.270,356.108,-76.624,-176.149,8.222,148.492
C06139=1190.266,356.356,-76.657,-176.147,8.226,148.493
C06140=1190.262,356.604,-76.690,-176.145,8.229,148.493
C06141=1190.259,356.851,-76.724,-176.143,8.232,148.493
C06142=1190.254,357.099,-76.758,-176.141,8.236,148.494
C06143=1190.249,357.347,-76.791,-176.139,8.239,148.494
C06144=1190.246,357.594,-76.825,-176.137,8.243,148.494
C06145=1190.242,357.842,-76.858,-176.135,8.246,148.494
C06146=1190.237,358.090,-76.891,-176.133,8.249,148.495
C06147=1190.234,358.338,-76.925,-176.131,8.252,148.495
C06148=1190.229,358.585,-76.959,-176.129,8.256,148.496
C06149=1190.225,358.833,-76.993,-176.127,8.259,148.496
C06150=1190.221,359.080,-77.026,-176.125,8.263,148.496
C06151=1190.217,359.328,-77.060,-176.123,8.266,148.496
C06152=1190.214,359.576,-77.093,-176.121,8.270,148.497
C06153=1190.209,359.824,-77.128,-176.120,8.272,148.497
C06154=1190.205,360.072,-77.161,-176.118,8.276,148.497
C06155=1190.201,360.319,-77.195,-176.116,8.280,148.498
C06156=1190.197,360.566,-77.228,-176.114,8.283,148.498
C06157=1190.193,360.815,-77.262,-176.112,8.286,148.499
C06158=1190.189,361.062,-77.296,-176.110,8.289,148.499
C06159=1190.185,361.310,-77.329,-176.108,8.293,148.499
C06160=1190.181,361.557,-77.363,-176.107,8.296,148.500
C06161=1190.177,361.806,-77.397,-176.104,8.300,148.500
C06162=1190.173,362.053,-77.431,-176.103,8.303,148.500
C06163=1190.169,362.301,-77.464,-176.101,8.306,148.501
C06164=1190.164,362.548,-77.498,-176.099,8.309,148.501
C06165=1190.161,362.797,-77.532,-176.097,8.313,148.501
C06166=1190.157,363.044,-77.566,-176.095,8.317,148.502
C06167=1190.153,363.291,-77.599,-176.094,8.319,148.502
C06168=1190.148,363.539,-77.633,-176.092,8.323,148.502
C06169=1190.145,363.787,-77.668,-176.090,8.326,148.503
C06170=1190.141,364.034,-77.701,-176.088,8.330,148.503
C06171=1190.136,364.282,-77.735,-176.087,8.333,148.504
C06172=1190.132,364.530,-77.768,-176.085,8.336,148.504
C06173=1190.128,364.778,-77.803,-176.084,8.340,148.504
C06174=1190.124,365.025,-77.837,-176.081,8.343,148.505
C06175=1190.120,365.272,-77.870,-176.080,8.346,148.505
C06176=1190.116,365.521,-77.905,-176.078,8.350,148.506
C06177=1190.112,365.768,-77.939,-176.076,8.353,148.506
C06178=1190.108,366.050,-77.977,-176.075,8.357,148.506
C06179=1190.103,366.330,-78.016,-176.073,8.361,148.507
C06180=1190.099,366.612,-78.055,-176.071,8.364,148.507
C06181=1190.093,366.892,-78.094,-176.069,8.368,148.508
C06182=1190.090,367.140,-78.127,-176.068,8.372,148.508
C06183=1190.085,367.388,-78.162,-176.066,8.375,148.509
C06184=1190.081,367.635,-78.195,-176.064,8.378,148.509
C06185=1190.078,367.883,-78.229,-176.063,8.382,148.509
C06186=1190.074,368.131,-78.264,-176.061,8.385,148.510
C06187=1190.070,368.378,-78.298,-176.060,8.388,148.510
C06188=1190.065,368.626,-78.332,-176.058,8.392,148.511
C06189=1190.062,368.874,-78.366,-176.057,8.394,148.511
C06190=1190.057,369.121,-78.400,-176.055,8.398,148.512
C06191=1190.054,369.369,-78.435,-176.053,8.402,148.512
C06192=1190.049,369.616,-78.469,-176.052,8.405,148.512
C06193=1190.045,369.864,-78.502,-176.050,8.408,148.513
C06194=1190.041,370.112,-78.537,-176.049,8.411,148.513
C06195=1190.037,370.359,-78.571,-176.047,8.415,148.514
C06196=1190.033,370.607,-78.606,-176.046,8.418,148.514
C06197=1190.029,370.855,-78.640,-176.045,8.422,148.515
C06198=1190.025,371.102,-78.674,-176.043,8.425,148.515
C06199=1190.021,371.350,-78.709,-176.042,8.428,148.516
C06200=1190.017,371.597,-78.743,-176.040,8.432,148.516
C06201=1190.013,371.845,-78.777,-176.039,8.434,148.516
C06202=1190.009,372.092,-78.812,-176.037,8.438,148.517
C06203=1190.005,372.340,-78.846,-176.036,8.441,148.517
C06204=1190.001,372.588,-78.881,-176.034,8.445,148.518
C06205=1189.997,372.835,-78.915,-176.034,8.448,148.518
C06206=1189.992,373.082,-78.949,-176.032,8.451,148.519
C06207=1189.989,373.330,-78.984,-176.030,8.454,148.519
C06208=1189.985,373.578,-79.018,-176.030,8.457,148.520
C06209=1189.981,373.826,-79.053,-176.028,8.461,148.520
C06210=1189.977,374.073,-79.087,-176.027,8.464,148.521
C06211=1189.973,374.321,-79.122,-176.025,8.468,148.521
C06212=1189.969,374.568,-79.155,-176.024,8.471,148.522
C06213=1189.965,374.816,-79.190,-176.022,8.474,148.522
C06214=1189.961,375.064,-79.225,-176.021,8.477,148.523
C06215=1189.957,375.311,-79.259,-176.020,8.480,148.523
C06216=1189.953,375.559,-79.293,-176.019,8.484,148.524
C06217=1189.948,375.806,-79.328,-176.018,8.487,148.524
C06218=1189.945,376.054,-79.362,-176.017,8.490,148.525
C06219=1189.940,376.302,-79.397,-176.015,8.494,148.525
C06220=1189.936,376.550,-79.431,-176.014,8.497,148.526
C06221=1189.933,376.796,-79.466,-176.013,8.499,148.526
C06222=1189.929,377.044,-79.501,-176.012,8.503,148.527
C06223=1189.924,377.292,-79.535,-176.010,8.506,148.527
C06224=1189.920,377.540,-79.570,-176.010,8.509,148.528
C06225=1189.917,377.787,-79.604,-176.008,8.513,148.528
C06226=1189.913,378.035,-79.639,-176.007,8.516,148.529
C06227=1189.908,378.282,-79.674,-176.006,8.519,148.529
C06228=1189.904,378.529,-79.708,-176.005,8.522,148.530
C06229=1189.900,378.777,-79.743,-176.004,8.526,148.530
C06230=1189.896,379.024,-79.777,-176.003,8.529,148.531
C06231=1189.892,379.273,-79.812,-176.002,8.532,148.531
C06232=1189.888,379.519,-79.847,-176.001,8.535,148.532
C06233=1189.884,379.767,-79.881,-176.000,8.538,148.533
C06234=1189.880,380.015,-79.916,-175.999,8.541,148.533
C06235=1189.876,380.262,-79.951,-175.997,8.545,148.534
C06236=1189.872,380.510,-79.986,-175.997,8.548,148.534
C06237=1189.868,380.757,-80.020,-175.995,8.551,148.535
C06238=1189.864,381.005,-80.055,-175.994,8.554,148.535
C06239=1189.860,381.252,-80.090,-175.994,8.557,148.536
C06240=1189.856,381.500,-80.125,-175.993,8.560,148.536
C06241=1189.852,381.748,-80.159,-175.992,8.563,148.537
C06242=1189.849,381.995,-80.194,-175.991,8.566,148.537
C06243=1189.844,382.242,-80.229,-175.990,8.569,148.538
C06244=1189.840,382.491,-80.264,-175.989,8.572,148.538
C06245=1189.836,382.737,-80.299,-175.988,8.576,148.539
C06246=1189.832,382.985,-80.334,-175.987,8.579,148.540
C06247=1189.827,383.233,-80.368,-175.986,8.582,148.540
C06248=1189.824,383.480,-80.403,-175.985,8.585,148.541
C06249=1189.820,383.728,-80.438,-175.985,8.587,148.541
C06250=1189.816,383.975,-80.473,-175.984,8.590,148.542
C06251=1189.812,384.223,-80.508,-175.983,8.593,148.542
C06252=1189.808,384.471,-80.542,-175.982,8.596,148.543
C06253=1189.804,384.718,-80.578,-175.982,8.599,148.543
C06254=1189.799,384.965,-80.612,-175.981,8.603,148.544
C06255=1189.797,385.213,-80.647,-175.980,8.606,148.545
C06256=1189.793,385.461,-80.682,-175.979,8.609,148.545
C06257=1189.788,385.708,-80.717,-175.978,8.612,148.546
C06258=1189.784,385.956,-80.752,-175.978,8.615,148.546
C06259=1189.780,386.203,-80.787,-175.977,8.617,148.547
C06260=1189.776,386.451,-80.822,-175.977,8.620,148.548
C06261=1189.772,386.699,-80.857,-175.976,8.623,148.548
C06262=1189.768,386.946,-80.892,-175.975,8.627,148.549
C06263=1189.764,387.194,-80.927,-175.974,8.630,148.549
C06264=1189.760,387.440,-80.962,-175.974,8.632,148.550
C06265=1189.756,387.689,-80.997,-175.973,8.635,148.550
C06266=1189.753,387.936,-81.032,-175.972,8.638,148.551
C06267=1189.748,388.183,-81.067,-175.971,8.641,148.552
C06268=1189.745,388.431,-81.102,-175.971,8.643,148.552
C06269=1189.740,388.677,-81.137,-175.970,8.647,148.553
C06270=1189.736,388.926,-81.172,-175.970,8.650,148.553
C06271=1189.733,389.173,-81.208,-175.970,8.652,148.554
C06272=1189.728,389.421,-81.242,-175.969,8.655,148.555
C06273=1189.724,389.668,-81.278,-175.969,8.658,148.555
C06274=1189.720,389.916,-81.312,-175.968,8.661,148.556
C06275=1189.716,390.163,-81.348,-175.967,8.664,148.556
C06276=1189.712,390.410,-81.383,-175.967,8.666,148.557
C06277=1189.709,390.659,-81.418,-175.966,8.669,148.557
C06278=1189.704,390.905,-81.453,-175.966,8.672,148.558
C06279=1189.700,391.153,-81.488,-175.966,8.675,148.559
C06280=1189.696,391.400,-81.523,-175.965,8.678,148.559
C06281=1189.692,391.648,-81.559,-175.964,8.680,148.560
C06282=1189.688,391.932,-81.599,-175.964,8.684,148.561
C06283=1189.683,392.215,-81.640,-175.963,8.687,148.561
C06284=1189.679,392.499,-81.679,-175.963,8.690,148.562
C06285=1189.674,392.782,-81.720,-175.963,8.692,148.562
C06286=1189.670,393.030,-81.754,-175.962,8.695,148.563
C06287=1189.667,393.277,-81.790,-175.962,8.698,148.564
C06288=1189.662,393.524,-81.825,-175.961,8.701,148.564
C06289=1189.658,393.772,-81.860,-175.961,8.703,148.565
C06290=1189.655,394.020,-81.895,-175.960,8.706,148.565
C06291=1189.650,394.266,-81.931,-175.960,8.709,148.566
C06292=1189.646,394.514,-81.965,-175.960,8.711,148.567
C06293=1189.643,394.762,-82.001,-175.959,8.714,148.567
C06294=1189.639,395.009,-82.037,-175.959,8.717,148.568
C06295=1189.634,395.257,-82.072,-175.959,8.719,148.568
C06296=1189.630,395.505,-82.107,-175.958,8.722,148.569
C06297=1189.626,395.752,-82.143,-175.958,8.725,148.570
C06298=1189.622,395.999,-82.178,-175.958,8.727,148.570
C06299=1189.618,396.247,-82.213,-175.957,8.730,148.571
C06300=1189.615,396.495,-82.248,-175.957,8.732,148.571
C06301=1189.610,396.741,-82.283,-175.957,8.735,148.572
C06302=1189.607,396.989,-82.319,-175.957,8.737,148.573
C06303=1189.603,397.237,-82.354,-175.956,8.740,148.573
C06304=1189.598,397.484,-82.389,-175.956,8.742,148.574
C06305=1189.595,397.731,-82.425,-175.956,8.745,148.574
C06306=1189.591,397.979,-82.460,-175.956,8.747,148.575
C06307=1189.587,398.226,-82.495,-175.955,8.750,148.576
C06308=1189.582,398.474,-82.531,-175.955,8.753,148.576
C06309=1189.578,398.722,-82.566,-175.955,8.755,148.577
C06310=1189.575,398.969,-82.602,-175.955,8.757,148.577
C06311=1189.571,399.216,-82.637,-175.955,8.760,148.578
C06312=1189.567,399.464,-82.672,-175.954,8.762,148.578
C06313=1189.563,399.712,-82.707,-175.953,8.765,148.579
C06314=1189.559,399.958,-82.743,-175.954,8.768,148.580
C06315=1189.555,400.206,-82.778,-175.953,8.770,148.580
C06316=1189.551,400.453,-82.814,-175.953,8.772,148.581
C06317=1189.547,400.702,-82.849,-175.953,8.774,148.581
C06318=1189.542,400.949,-82.884,-175.953,8.777,148.582
C06319=1189.539,401.196,-82.920,-175.953,8.779,148.582
C06320=1189.535,401.444,-82.955,-175.953,8.782,148.583
C06321=1189.531,401.690,-82.991,-175.952,8.784,148.584
C06322=1189.527,401.938,-83.026,-175.952,8.786,148.584
C06323=1189.523,402.185,-83.062,-175.952,8.789,148.585
C06324=1189.519,402.434,-83.097,-175.951,8.792,148.585
C06325=1189.514,402.681,-83.132,-175.951,8.794,148.586
C06326=1189.511,402.928,-83.168,-175.951,8.796,148.586
C06327=1189.507,403.176,-83.203,-175.951,8.799,148.587
C06328=1189.503,403.423,-83.239,-175.951,8.801,148.588
C06329=1189.499,403.670,-83.274,-175.951,8.803,148.588
C06330=1189.495,403.918,-83.310,-175.950,8.806,148.589
C06331=1189.491,404.165,-83.346,-175.950,8.808,148.589
C06332=1189.487,404.413,-83.381,-175.950,8.810,148.590
C06333=1189.483,404.660,-83.416,-175.950,8.813,148.591
C06334=1189.479,404.908,-83.451,-175.950,8.814,148.591
C06335=1189.476,405.155,-83.487,-175.950,8.816,148.591
C06336=1189.471,405.403,-83.523,-175.950,8.819,148.592
C06337=1189.467,405.650,-83.558,-175.950,8.821,148.593
C06338=1189.463,405.897,-83.594,-175.950,8.824,148.593
C06339=1189.460,406.145,-83.629,-175.950,8.826,148.594
C06340=1189.456,406.392,-83.665,-175.949,8.828,148.594
C06341=1189.451,406.639,-83.701,-175.949,8.830,148.595
C06342=1189.447,406.887,-83.736,-175.949,8.833,148.596
C06343=1189.444,407.134,-83.772,-175.949,8.835,148.596
C06344=1189.440,407.382,-83.807,-175.949,8.837,148.597
C06345=1189.436,407.629,-83.843,-175.949,8.839,148.597
C06346=1189.431,407.876,-83.879,-175.949,8.841,148.598
C06347=1189.428,408.124,-83.914,-175.949,8.843,148.598
C06348=1189.424,408.371,-83.950,-175.948,8.846,148.599
C06349=1189.420,408.619,-83.985,-175.949,8.848,148.599
C06350=1189.416,408.866,-84.020,-175.948,8.850,148.600
C06351=1189.412,409.114,-84.057,-175.949,8.852,148.600
C06352=1189.408,409.361,-84.092,-175.948,8.854,148.601
C06353=1189.404,409.609,-84.128,-175.948,8.856,148.601
C06354=1189.401,409.856,-84.163,-175.948,8.859,148.602
C06355=1189.396,410.103,-84.198,-175.948,8.861,148.602
C06356=1189.392,410.351,-84.235,-175.947,8.863,148.603
C06357=1189.388,410.598,-84.270,-175.948,8.865,148.604
C06358=1189.385,410.846,-84.306,-175.948,8.867,148.604
C06359=1189.381,411.093,-84.341,-175.948,8.870,148.605
C06360=1189.376,411.340,-84.377,-175.947,8.872,148.605
C06361=1189.372,411.588,-84.413,-175.948,8.873,148.606
C06362=1189.369,411.835,-84.448,-175.947,8.875,148.606
C06363=1189.365,412.083,-84.484,-175.947,8.878,148.607
C06364=1189.361,412.331,-84.520,-175.947,8.880,148.607
C06365=1189.356,412.577,-84.555,-175.947,8.881,148.608
C06366=1189.353,412.825,-84.590,-175.947,8.884,148.608
C06367=1189.349,413.072,-84.626,-175.947,8.886,148.609
C06368=1189.345,413.320,-84.662,-175.946,8.888,148.609
C06369=1189.341,413.568,-84.698,-175.947,8.890,148.610
C06370=1189.337,413.814,-84.733,-175.947,8.892,148.610
C06371=1189.332,414.062,-84.769,-175.947,8.894,148.611
C06372=1189.329,414.310,-84.805,-175.947,8.896,148.611
C06373=1189.325,414.557,-84.840,-175.947,8.898,148.612
C06374=1189.321,414.805,-84.876,-175.946,8.900,148.613
C06375=1189.317,415.051,-84.912,-175.947,8.902,148.613
C06376=1189.313,415.299,-84.948,-175.947,8.904,148.613
C06377=1189.309,415.546,-84.983,-175.946,8.906,148.614
C06378=1189.302,415.940,-85.040,-175.946,8.909,148.615
C06379=1189.299,416.334,-85.097,-175.946,8.912,148.616
C06380=1189.299,416.728,-85.153,-175.946,8.916,148.616
C06381=1189.302,417.121,-85.209,-175.946,8.918,148.617
C06382=1188.880,417.122,-85.250,-175.949,8.929,148.621
C06383=1188.877,416.725,-85.194,-175.949,8.926,148.620
C06384=1188.877,416.329,-85.137,-175.949,8.923,148.619
C06385=1188.881,415.933,-85.080,-175.949,8.920,148.618
C06386=1188.887,415.536,-85.023,-175.949,8.917,148.618
C06387=1188.892,415.288,-84.986,-175.950,8.915,148.617
C06388=1188.895,415.040,-84.951,-175.949,8.913,148.617
C06389=1188.900,414.794,-84.916,-175.950,8.911,148.616
C06390=1188.904,414.546,-84.880,-175.950,8.909,148.616
C06391=1188.908,414.298,-84.844,-175.950,8.907,148.615
C06392=1188.911,414.051,-84.808,-175.950,8.905,148.615
C06393=1188.915,413.804,-84.772,-175.950,8.903,148.614
C06394=1188.920,413.557,-84.736,-175.950,8.901,148.614
C06395=1188.923,413.309,-84.701,-175.950,8.899,148.613
C06396=1188.927,413.062,-84.665,-175.950,8.897,148.612
C06397=1188.931,412.814,-84.629,-175.950,8.894,148.612
C06398=1188.935,412.566,-84.594,-175.950,8.892,148.611
C06399=1188.939,412.320,-84.559,-175.950,8.891,148.611
C06400=1188.943,412.072,-84.523,-175.950,8.888,148.610
C06401=1188.947,411.824,-84.487,-175.950,8.886,148.610
C06402=1188.951,411.577,-84.451,-175.950,8.885,148.609
C06403=1188.955,411.329,-84.416,-175.950,8.882,148.609
C06404=1188.959,411.082,-84.381,-175.951,8.880,148.608
C06405=1188.963,410.835,-84.344,-175.951,8.878,148.608
C06406=1188.967,410.587,-84.309,-175.951,8.876,148.607
C06407=1188.971,410.340,-84.273,-175.950,8.874,148.607
C06408=1188.974,410.092,-84.238,-175.951,8.872,148.606
C06409=1188.979,409.845,-84.202,-175.951,8.869,148.606
C06410=1188.983,409.598,-84.166,-175.951,8.867,148.605
C06411=1188.987,409.350,-84.131,-175.951,8.866,148.605
C06412=1188.990,409.103,-84.095,-175.951,8.863,148.604
C06413=1188.995,408.855,-84.059,-175.951,8.861,148.604
C06414=1188.999,408.608,-84.024,-175.951,8.859,148.603
C06415=1189.003,408.360,-83.988,-175.951,8.856,148.602
C06416=1189.006,408.113,-83.953,-175.952,8.854,148.602
C06417=1189.010,407.865,-83.917,-175.951,8.853,148.601
C06418=1189.014,407.618,-83.881,-175.952,8.850,148.601
C06419=1189.019,407.371,-83.846,-175.952,8.848,148.600
C06420=1189.022,407.123,-83.810,-175.952,8.846,148.600
C06421=1189.026,406.876,-83.775,-175.952,8.843,148.599
C06422=1189.030,406.628,-83.739,-175.952,8.841,148.598
C06423=1189.035,406.381,-83.704,-175.952,8.839,148.598
C06424=1189.038,406.134,-83.668,-175.953,8.836,148.597
C06425=1189.042,405.886,-83.633,-175.952,8.835,148.597
C06426=1189.046,405.639,-83.597,-175.952,8.832,148.596
C06427=1189.050,405.392,-83.562,-175.952,8.830,148.596
C06428=1189.054,405.144,-83.526,-175.953,8.828,148.595
C06429=1189.058,404.897,-83.490,-175.953,8.826,148.595
C06430=1189.062,404.649,-83.455,-175.953,8.823,148.594
C06431=1189.065,404.402,-83.419,-175.953,8.821,148.593
C06432=1189.070,404.155,-83.384,-175.953,8.819,148.593
C06433=1189.074,403.907,-83.348,-175.954,8.816,148.592
C06434=1189.078,403.659,-83.313,-175.954,8.814,148.592
C06435=1189.082,403.411,-83.277,-175.954,8.811,148.591
C06436=1189.086,403.165,-83.242,-175.954,8.809,148.591
C06437=1189.090,402.917,-83.207,-175.954,8.807,148.590
C06438=1189.093,402.670,-83.171,-175.954,8.805,148.590
C06439=1189.097,402.423,-83.136,-175.955,8.802,148.589
C06440=1189.102,402.175,-83.100,-175.954,8.800,148.588
C06441=1189.106,401.927,-83.064,-175.955,8.798,148.588
C06442=1189.109,401.680,-83.029,-175.955,8.795,148.587
C06443=1189.114,401.433,-82.994,-175.955,8.793,148.587
C06444=1189.117,401.185,-82.959,-175.955,8.790,148.586
C06445=1189.121,400.938,-82.923,-175.955,8.788,148.585
C06446=1189.125,400.690,-82.887,-175.955,8.786,148.585
C06447=1189.130,400.443,-82.852,-175.956,8.783,148.584
C06448=1189.133,400.195,-82.816,-175.956,8.780,148.584
C06449=1189.137,399.947,-82.781,-175.956,8.778,148.583
C06450=1189.141,399.700,-82.746,-175.957,8.776,148.583
C06451=1189.145,399.453,-82.711,-175.957,8.773,148.582
C06452=1189.149,399.206,-82.675,-175.957,8.771,148.581
C06453=1189.153,398.958,-82.640,-175.957,8.769,148.581
C06454=1189.158,398.711,-82.604,-175.958,8.766,148.580
C06455=1189.162,398.463,-82.569,-175.958,8.763,148.580
C06456=1189.165,398.215,-82.533,-175.958,8.761,148.579
C06457=1189.169,397.968,-82.498,-175.958,8.758,148.578
C06458=1189.173,397.721,-82.463,-175.958,8.756,148.578
C06459=1189.177,397.473,-82.428,-175.959,8.753,148.577
C06460=1189.181,397.225,-82.392,-175.959,8.751,148.577
C06461=1189.185,396.979,-82.357,-175.959,8.748,148.576
C06462=1189.189,396.731,-82.322,-175.959,8.746,148.576
C06463=1189.192,396.484,-82.286,-175.960,8.743,148.575
C06464=1189.197,396.236,-82.252,-175.960,8.740,148.574
C06465=1189.201,395.988,-82.215,-175.960,8.738,148.574
C06466=1189.205,395.741,-82.180,-175.960,8.736,148.573
C06467=1189.210,395.493,-82.145,-175.961,8.733,148.573
C06468=1189.213,395.246,-82.110,-175.961,8.730,148.572
C06469=1189.217,394.998,-82.074,-175.961,8.728,148.571
C06470=1189.221,394.751,-82.039,-175.962,8.725,148.571
C06471=1189.225,394.504,-82.004,-175.962,8.722,148.570
C06472=1189.229,394.256,-81.969,-175.963,8.719,148.569
C06473=1189.232,394.009,-81.933,-175.963,8.717,148.569
C06474=1189.237,393.761,-81.899,-175.963,8.715,148.568
C06475=1189.241,393.514,-81.863,-175.964,8.711,148.568
C06476=1189.244,393.266,-81.828,-175.964,8.709,148.567
C06477=1189.249,393.019,-81.792,-175.965,8.706,148.567
C06478=1189.253,392.771,-81.758,-175.965,8.704,148.566
C06479=1189.257,392.488,-81.717,-175.966,8.700,148.565
C06480=1189.262,392.204,-81.677,-175.966,8.697,148.565
C06481=1189.266,391.920,-81.636,-175.967,8.694,148.564
C06482=1189.272,391.637,-81.596,-175.967,8.691,148.563
C06483=1189.275,391.390,-81.561,-175.967,8.688,148.563
C06484=1189.279,391.142,-81.525,-175.968,8.686,148.562
C06485=1189.283,390.895,-81.491,-175.968,8.683,148.562
C06486=1189.287,390.647,-81.455,-175.969,8.680,148.561
C06487=1189.291,390.399,-81.420,-175.969,8.677,148.560
C06488=1189.295,390.152,-81.385,-175.970,8.674,148.560
C06489=1189.298,389.905,-81.350,-175.970,8.672,148.559
C06490=1189.302,389.657,-81.315,-175.971,8.669,148.559
C06491=1189.306,389.410,-81.280,-175.972,8.666,148.558
C06492=1189.310,389.162,-81.245,-175.972,8.663,148.557
C06493=1189.315,388.915,-81.210,-175.972,8.660,148.557
C06494=1189.319,388.667,-81.175,-175.973,8.658,148.556
C06495=1189.322,388.420,-81.140,-175.973,8.655,148.556
C06496=1189.327,388.173,-81.105,-175.974,8.652,148.555
C06497=1189.331,387.925,-81.070,-175.975,8.648,148.554
C06498=1189.334,387.677,-81.034,-175.975,8.646,148.554
C06499=1189.339,387.430,-81.000,-175.976,8.643,148.553
C06500=1189.342,387.182,-80.964,-175.977,8.640,148.553
C06501=1189.347,386.935,-80.930,-175.978,8.637,148.552
C06502=1189.351,386.687,-80.894,-175.978,8.635,148.552
C06503=1189.355,386.439,-80.859,-175.979,8.632,148.551
C06504=1189.359,386.192,-80.824,-175.980,8.628,148.550
C06505=1189.362,385.945,-80.790,-175.980,8.625,148.550
C06506=1189.366,385.698,-80.755,-175.981,8.622,148.549
C06507=1189.370,385.450,-80.720,-175.981,8.620,148.549
C06508=1189.374,385.202,-80.684,-175.982,8.617,148.548
C06509=1189.379,384.955,-80.650,-175.983,8.614,148.548
C06510=1189.383,384.707,-80.615,-175.984,8.611,148.547
C06511=1189.387,384.460,-80.580,-175.985,8.608,148.546
C06512=1189.391,384.212,-80.545,-175.985,8.604,148.546
C06513=1189.395,383.965,-80.510,-175.986,8.601,148.545
C06514=1189.398,383.717,-80.476,-175.987,8.598,148.545
C06515=1189.402,383.469,-80.441,-175.988,8.595,148.544
C06516=1189.407,383.222,-80.406,-175.989,8.592,148.543
C06517=1189.411,382.974,-80.371,-175.989,8.589,148.543
C06518=1189.415,382.727,-80.336,-175.990,8.586,148.542
C06519=1189.419,382.479,-80.301,-175.991,8.583,148.542
C06520=1189.423,382.232,-80.267,-175.992,8.580,148.541
C06521=1189.426,381.985,-80.231,-175.993,8.577,148.541
C06522=1189.430,381.736,-80.197,-175.994,8.574,148.540
C06523=1189.435,381.489,-80.162,-175.995,8.571,148.540
C06524=1189.438,381.242,-80.126,-175.995,8.568,148.539
C06525=1189.443,380.994,-80.092,-175.997,8.565,148.539
C06526=1189.446,380.746,-80.058,-175.998,8.561,148.538
C06527=1189.450,380.500,-80.023,-175.999,8.558,148.537
C06528=1189.454,380.251,-79.988,-176.000,8.555,148.537
C06529=1189.459,380.004,-79.953,-176.001,8.552,148.536
C06530=1189.463,379.756,-79.918,-176.002,8.549,148.536
C06531=1189.467,379.509,-79.884,-176.002,8.546,148.535
C06532=1189.471,379.261,-79.849,-176.004,8.542,148.535
C06533=1189.475,379.014,-79.815,-176.005,8.539,148.534
C06534=1189.479,378.766,-79.780,-176.006,8.536,148.534
C06535=1189.483,378.519,-79.745,-176.007,8.533,148.533
C06536=1189.487,378.271,-79.710,-176.008,8.530,148.533
C06537=1189.491,378.024,-79.676,-176.009,8.526,148.532
C06538=1189.495,377.776,-79.641,-176.011,8.523,148.532
C06539=1189.499,377.529,-79.606,-176.011,8.520,148.531
C06540=1189.503,377.281,-79.572,-176.013,8.517,148.531
C06541=1189.507,377.034,-79.537,-176.014,8.513,148.530
C06542=1189.510,376.786,-79.503,-176.015,8.511,148.530
C06543=1189.515,376.538,-79.468,-176.017,8.507,148.529
C06544=1189.519,376.290,-79.434,-176.017,8.504,148.528
C06545=1189.523,376.043,-79.399,-176.019,8.501,148.528
C06546=1189.526,375.796,-79.364,-176.020,8.497,148.527
C06547=1189.531,375.548,-79.330,-176.021,8.494,148.527
C06548=1189.535,375.300,-79.295,-176.022,8.491,148.527
C06549=1189.539,375.053,-79.261,-176.024,8.487,148.526
C06550=1189.543,374.806,-79.227,-176.025,8.485,148.526
C06551=1189.547,374.557,-79.192,-176.026,8.481,148.525
C06552=1189.551,374.310,-79.158,-176.028,8.478,148.525
C06553=1189.555,374.062,-79.123,-176.028,8.475,148.524
C06554=1189.559,373.815,-79.089,-176.030,8.471,148.524
C06555=1189.563,373.567,-79.054,-176.031,8.468,148.523
C06556=1189.567,373.319,-79.020,-176.033,8.464,148.523
C06557=1189.571,373.072,-78.986,-176.034,8.462,148.522
C06558=1189.575,372.824,-78.951,-176.036,8.458,148.522
C06559=1189.580,372.577,-78.917,-176.037,8.455,148.521
C06560=1189.583,372.329,-78.882,-176.038,8.451,148.521
C06561=1189.588,372.082,-78.848,-176.040,8.448,148.520
C06562=1189.591,371.834,-78.814,-176.041,8.445,148.520
C06563=1189.595,371.586,-78.779,-176.042,8.442,148.519
C06564=1189.599,371.339,-78.745,-176.044,8.438,148.519
C06565=1189.603,371.091,-78.711,-176.045,8.435,148.519
C06566=1189.608,370.844,-78.676,-176.047,8.432,148.518
C06567=1189.611,370.596,-78.642,-176.048,8.429,148.517
C06568=1189.616,370.349,-78.607,-176.050,8.425,148.517
C06569=1189.619,370.101,-78.574,-176.051,8.422,148.517
C06570=1189.623,369.853,-78.539,-176.053,8.418,148.516
C06571=1189.628,369.606,-78.506,-176.055,8.415,148.516
C06572=1189.632,369.358,-78.471,-176.056,8.412,148.515
C06573=1189.635,369.110,-78.437,-176.058,8.408,148.515
C06574=1189.640,368.863,-78.402,-176.058,8.405,148.514
C06575=1189.643,368.615,-78.368,-176.060,8.402,148.514
C06576=1189.648,368.368,-78.334,-176.062,8.398,148.514
C06577=1189.652,368.120,-78.301,-176.063,8.395,148.513
C06578=1189.656,367.872,-78.266,-176.065,8.392,148.513
C06579=1189.660,367.625,-78.232,-176.066,8.389,148.512
C06580=1189.664,367.377,-78.197,-176.068,8.385,148.512
C06581=1189.668,367.129,-78.164,-176.070,8.382,148.511
C06582=1189.672,366.881,-78.129,-176.071,8.379,148.511
C06583=1189.677,366.601,-78.091,-176.073,8.374,148.511
C06584=1189.681,366.320,-78.052,-176.075,8.371,148.510
C06585=1189.685,366.038,-78.013,-176.077,8.367,148.510
C06586=1189.690,365.757,-77.975,-176.079,8.363,148.509
C06587=1189.695,365.510,-77.941,-176.081,8.360,148.509
C06588=1189.698,365.262,-77.907,-176.082,8.356,148.508
C06589=1189.702,365.014,-77.874,-176.084,8.353,148.508
C06590=1189.707,364.767,-77.839,-176.086,8.350,148.508
C06591=1189.710,364.519,-77.805,-176.088,8.346,148.507
C06592=1189.714,364.271,-77.772,-176.090,8.343,148.507
C06593=1189.719,364.024,-77.737,-176.091,8.340,148.507
C06594=1189.723,363.777,-77.703,-176.093,8.336,148.506
C06595=1189.727,363.528,-77.669,-176.094,8.333,148.506
C06596=1189.731,363.281,-77.635,-176.097,8.329,148.505
C06597=1189.735,363.033,-77.602,-176.098,8.327,148.505
C06598=1189.739,362.785,-77.567,-176.100,8.323,148.505
C06599=1189.743,362.537,-77.534,-176.101,8.319,148.504
C06600=1189.747,362.290,-77.500,-176.104,8.316,148.504
C06601=1189.751,362.043,-77.466,-176.105,8.313,148.504
C06602=1189.755,361.794,-77.432,-176.107,8.310,148.503
C06603=1189.759,361.547,-77.398,-176.109,8.306,148.503
C06604=1189.763,361.299,-77.365,-176.111,8.303,148.502
C06605=1189.768,361.052,-77.331,-176.113,8.299,148.502
C06606=1189.771,360.803,-77.297,-176.114,8.297,148.502
C06607=1189.775,360.556,-77.264,-176.116,8.293,148.501
C06608=1189.779,360.309,-77.230,-176.118,8.290,148.501
C06609=1189.784,360.061,-77.197,-176.120,8.286,148.501
C06610=1189.788,359.813,-77.163,-176.122,8.282,148.500
C06611=1189.791,359.565,-77.129,-176.124,8.279,148.500
C06612=1189.795,359.318,-77.095,-176.125,8.276,148.500
C06613=1189.799,359.070,-77.062,-176.128,8.273,148.499
C06614=1189.804,358.822,-77.028,-176.129,8.269,148.499
C06615=1189.808,358.575,-76.994,-176.132,8.266,148.499
C06616=1189.811,358.327,-76.961,-176.133,8.262,148.498
C06617=1189.816,358.079,-76.928,-176.136,8.259,148.498
C06618=1189.819,357.832,-76.894,-176.138,8.255,148.498
C06619=1189.824,357.584,-76.860,-176.140,8.252,148.498
C06620=1189.828,357.336,-76.827,-176.141,8.249,148.497
C06621=1189.832,357.089,-76.793,-176.143,8.246,148.497
C06622=1189.836,356.840,-76.760,-176.145,8.243,148.497
C06623=1189.840,356.593,-76.726,-176.147,8.239,148.496
C06624=1189.844,356.345,-76.693,-176.150,8.236,148.496
C06625=1189.849,356.098,-76.659,-176.151,8.232,148.496
C06626=1189.853,355.850,-76.626,-176.154,8.229,148.495
C06627=1189.857,355.602,-76.593,-176.156,8.225,148.495
C06628=1189.861,355.354,-76.559,-176.157,8.223,148.495
C06629=1189.865,355.107,-76.526,-176.159,8.219,148.495
C06630=1189.868,354.859,-76.492,-176.162,8.216,148.494
C06631=1189.873,354.611,-76.459,-176.163,8.212,148.494
C06632=1189.877,354.363,-76.426,-176.166,8.209,148.494
C06633=1189.881,354.116,-76.393,-176.168,8.206,148.493
C06634=1189.885,353.868,-76.359,-176.170,8.202,148.493
C06635=1189.889,353.620,-76.326,-176.172,8.199,148.493
C06636=1189.893,353.372,-76.293,-176.174,8.195,148.493
C06637=1189.897,353.125,-76.260,-176.176,8.193,148.492
C06638=1189.902,352.877,-76.227,-176.178,8.189,148.492
C06639=1189.906,352.630,-76.192,-176.180,8.186,148.492
C06640=1189.910,352.382,-76.159,-176.182,8.183,148.491
C06641=1189.914,352.133,-76.126,-176.184,8.179,148.491
C06642=1189.918,351.886,-76.092,-176.186,8.176,148.491
C06643=1189.922,351.638,-76.059,-176.188,8.172,148.491
C06644=1189.926,351.390,-76.026,-176.191,8.169,148.490
C06645=1189.930,351.143,-75.994,-176.192,8.167,148.490
C06646=1189.934,350.895,-75.960,-176.195,8.163,148.490
C06647=1189.938,350.647,-75.927,-176.196,8.160,148.490
C06648=1189.942,350.399,-75.895,-176.199,8.156,148.489
C06649=1189.946,350.151,-75.862,-176.201,8.153,148.489
C06650=1189.951,349.904,-75.829,-176.203,8.150,148.489
C06651=1189.955,349.656,-75.795,-176.205,8.146,148.489
C06652=1189.959,349.408,-75.762,-176.208,8.143,148.488
C06653=1189.963,349.160,-75.729,-176.209,8.140,148.488
C06654=1189.967,348.913,-75.696,-176.211,8.137,148.488
C06655=1189.971,348.665,-75.663,-176.213,8.133,148.488
C06656=1189.975,348.417,-75.630,-176.216,8.130,148.487
C06657=1189.980,348.169,-75.597,-176.218,8.127,148.487
C06658=1189.984,347.921,-75.564,-176.220,8.124,148.487
C06659=1189.987,347.674,-75.531,-176.222,8.120,148.487
C06660=1189.992,347.426,-75.498,-176.225,8.117,148.487
C06661=1189.996,347.178,-75.465,-176.227,8.114,148.486
C06662=1190.000,346.930,-75.433,-176.228,8.111,148.486
C06663=1190.004,346.682,-75.400,-176.231,8.108,148.486
C06664=1190.008,346.434,-75.366,-176.233,8.104,148.486
C06665=1190.012,346.187,-75.334,-176.235,8.101,148.485
C06666=1190.016,345.939,-75.301,-176.237,8.098,148.485
C06667=1190.021,345.692,-75.269,-176.240,8.094,148.485
C06668=1190.025,345.444,-75.235,-176.242,8.091,148.485
C06669=1190.029,345.196,-75.202,-176.244,8.088,148.485
C06670=1190.033,344.948,-75.170,-176.246,8.085,148.484
C06671=1190.037,344.700,-75.137,-176.248,8.082,148.484
C06672=1190.041,344.453,-75.104,-176.250,8.079,148.484
C06673=1190.046,344.204,-75.072,-176.253,8.075,148.484
C06674=1190.050,343.957,-75.039,-176.255,8.072,148.484
C06675=1190.054,343.709,-75.007,-176.257,8.069,148.483
C06676=1190.058,343.461,-74.974,-176.259,8.065,148.483
C06677=1190.062,343.213,-74.940,-176.262,8.062,148.483
C06678=1190.067,342.965,-74.908,-176.263,8.060,148.483
C06679=1190.070,342.718,-74.876,-176.265,8.056,148.483
C06680=1190.075,342.470,-74.843,-176.268,8.053,148.482
C06681=1190.079,342.222,-74.810,-176.270,8.050,148.482
C06682=1190.083,341.974,-74.778,-176.273,8.047,148.482
C06683=1190.087,341.726,-74.745,-176.275,8.043,148.482
C06684=1190.091,341.478,-74.713,-176.277,8.040,148.482
C06685=1190.095,341.231,-74.680,-176.279,8.037,148.481
C06686=1190.100,340.983,-74.648,-176.281,8.034,148.481
C06687=1190.104,340.704,-74.611,-176.284,8.030,148.481
C06688=1190.109,340.426,-74.575,-176.286,8.027,148.481
C06689=1190.114,340.147,-74.538,-176.289,8.024,148.481
C06690=1190.118,339.868,-74.502,-176.292,8.019,148.480
C06691=1190.122,339.620,-74.469,-176.294,8.016,148.480
C06692=1190.126,339.372,-74.437,-176.296,8.013,148.480
C06693=1190.130,339.124,-74.404,-176.298,8.010,148.480
C06694=1190.135,338.877,-74.372,-176.301,8.007,148.480
C06695=1190.139,338.628,-74.340,-176.303,8.004,148.480
C06696=1190.143,338.381,-74.307,-176.305,8.001,148.479
C06697=1190.147,338.133,-74.275,-176.307,7.997,148.479
C06698=1190.151,337.885,-74.243,-176.309,7.994,148.479
C06699=1190.156,337.638,-74.210,-176.312,7.991,148.479
C06700=1190.159,337.390,-74.178,-176.314,7.988,148.479
C06701=1190.164,337.141,-74.146,-176.316,7.985,148.479
C06702=1190.168,336.893,-74.113,-176.318,7.982,148.478
C06703=1190.172,336.645,-74.081,-176.321,7.979,148.478
C06704=1190.177,336.398,-74.049,-176.323,7.975,148.478
C06705=1190.180,336.150,-74.017,-176.326,7.972,148.478
C06706=1190.185,335.901,-73.985,-176.328,7.969,148.478
C06707=1190.188,335.654,-73.952,-176.330,7.966,148.478
C06708=1190.192,335.407,-73.920,-176.332,7.963,148.478
C06709=1190.197,335.158,-73.888,-176.334,7.960,148.477
C06710=1190.201,334.910,-73.856,-176.337,7.957,148.477
C06711=1190.205,334.662,-73.824,-176.339,7.954,148.477
C06712=1190.209,334.415,-73.792,-176.342,7.950,148.477
C06713=1190.213,334.167,-73.759,-176.344,7.947,148.477
C06714=1190.217,333.919,-73.727,-176.347,7.944,148.477
C06715=1190.222,333.671,-73.695,-176.348,7.941,148.477
C06716=1190.226,333.423,-73.663,-176.350,7.938,148.476
C06717=1190.230,333.175,-73.632,-176.353,7.935,148.476
C06718=1190.234,332.927,-73.599,-176.355,7.932,148.476
C06719=1190.238,332.679,-73.568,-176.358,7.929,148.476
C06720=1190.242,332.431,-73.536,-176.360,7.925,148.476
C06721=1190.247,332.183,-73.503,-176.363,7.922,148.476
C06722=1190.251,331.936,-73.472,-176.365,7.920,148.476
C06723=1190.255,331.687,-73.439,-176.367,7.917,148.476
C06724=1190.259,331.439,-73.408,-176.369,7.913,148.475
C06725=1190.263,331.192,-73.376,-176.372,7.910,148.475
C06726=1190.268,330.944,-73.344,-176.374,7.907,148.475
C06727=1190.271,330.696,-73.312,-176.377,7.904,148.475
C06728=1190.276,330.448,-73.280,-176.379,7.901,148.475
C06729=1190.280,330.200,-73.248,-176.381,7.898,148.475
C06730=1190.284,329.953,-73.216,-176.384,7.895,148.475
C06731=1190.288,329.704,-73.185,-176.386,7.892,148.474
C06732=1190.292,329.456,-73.153,-176.388,7.889,148.474
C06733=1190.297,329.208,-73.121,-176.391,7.885,148.474
C06734=1190.301,328.960,-73.089,-176.393,7.882,148.474
C06735=1190.305,328.712,-73.058,-176.395,7.880,148.474
C06736=1190.309,328.465,-73.026,-176.397,7.877,148.474
C06737=1190.313,328.216,-72.994,-176.400,7.874,148.474
C06738=1190.318,327.969,-72.962,-176.402,7.870,148.474
C06739=1190.322,327.720,-72.931,-176.405,7.867,148.474
C06740=1190.325,327.472,-72.899,-176.407,7.864,148.473
C06741=1190.330,327.225,-72.867,-176.410,7.861,148.473
C06742=1190.334,326.977,-72.835,-176.412,7.858,148.473
C06743=1190.339,326.729,-72.805,-176.414,7.855,148.473
C06744=1190.343,326.481,-72.773,-176.417,7.852,148.473
C06745=1190.347,326.233,-72.741,-176.419,7.849,148.473
C06746=1190.351,325.985,-72.709,-176.422,7.846,148.473
C06747=1190.355,325.736,-72.678,-176.424,7.843,148.473
C06748=1190.360,325.489,-72.646,-176.426,7.840,148.473
C06749=1190.363,325.241,-72.614,-176.429,7.837,148.473
C06750=1190.368,324.993,-72.584,-176.431,7.834,148.473
C06751=1190.372,324.745,-72.552,-176.434,7.831,148.473
C06752=1190.376,324.498,-72.520,-176.436,7.828,148.472
C06753=1190.380,324.249,-72.489,-176.438,7.825,148.472
C06754=1190.384,324.002,-72.458,-176.440,7.822,148.472
C06755=1190.389,323.753,-72.426,-176.443,7.819,148.472
C06756=1190.393,323.505,-72.394,-176.445,7.816,148.472
C06757=1190.397,323.257,-72.363,-176.448,7.813,148.472
C06758=1190.402,323.009,-72.332,-176.450,7.809,148.472
C06759=1190.405,322.761,-72.300,-176.453,7.806,148.472
C06760=1190.410,322.513,-72.269,-176.455,7.804,148.472
C06761=1190.414,322.265,-72.237,-176.457,7.801,148.472
C06762=1190.418,322.017,-72.207,-176.460,7.798,148.472
C06763=1190.422,321.769,-72.175,-176.462,7.795,148.471
C06764=1190.427,321.521,-72.144,-176.465,7.792,148.471
C06765=1190.430,321.273,-72.112,-176.468,7.789,148.471
C06766=1190.435,321.025,-72.081,-176.469,7.786,148.471
C06767=1190.439,320.777,-72.050,-176.472,7.783,148.471
C06768=1190.443,320.529,-72.019,-176.474,7.780,148.471
C06769=1190.447,320.281,-71.988,-176.477,7.777,148.471
C06770=1190.452,320.033,-71.956,-176.480,7.774,148.471
C06771=1190.456,319.785,-71.925,-176.482,7.770,148.471
C06772=1190.460,319.537,-71.894,-176.484,7.768,148.471
C06773=1190.464,319.289,-71.863,-176.486,7.765,148.471
C06774=1190.468,319.041,-71.832,-176.489,7.762,148.471
C06775=1190.473,318.793,-71.800,-176.492,7.759,148.471
C06776=1190.476,318.545,-71.770,-176.494,7.756,148.471
C06777=1190.481,318.297,-71.739,-176.497,7.753,148.471
C06778=1190.485,318.048,-71.708,-176.499,7.750,148.471
C06779=1190.489,317.801,-71.676,-176.501,7.747,148.470
C06780=1190.494,317.553,-71.646,-176.504,7.744,148.470
C06781=1190.498,317.304,-71.614,-176.506,7.741,148.470
C06782=1190.502,317.057,-71.583,-176.509,7.738,148.470
C06783=1190.506,316.808,-71.552,-176.511,7.735,148.470
C06784=1190.510,316.561,-71.522,-176.513,7.732,148.470
C06785=1190.514,316.313,-71.491,-176.516,7.729,148.470
C06786=1190.518,316.064,-71.460,-176.518,7.726,148.470
C06787=1190.523,315.817,-71.428,-176.521,7.723,148.470
C06788=1190.527,315.569,-71.398,-176.523,7.721,148.470
C06789=1190.531,315.320,-71.366,-176.525,7.718,148.470
C06790=1190.535,315.073,-71.336,-176.528,7.715,148.470
C06791=1190.540,314.796,-71.301,-176.530,7.711,148.470
C06792=1190.545,314.519,-71.267,-176.534,7.707,148.470
C06793=1190.549,314.243,-71.233,-176.536,7.704,148.470
C06794=1190.554,313.967,-71.198,-176.539,7.701,148.470
C06795=1190.558,313.718,-71.167,-176.542,7.698,148.470
C06796=1190.563,313.470,-71.137,-176.544,7.695,148.470
C06797=1190.567,313.222,-71.106,-176.546,7.693,148.470
C06798=1190.571,312.975,-71.076,-176.549,7.690,148.470
C06799=1190.575,312.726,-71.045,-176.551,7.687,148.469
C06800=1190.580,312.478,-71.014,-176.554,7.684,148.469
C06801=1190.584,312.231,-70.984,-176.557,7.681,148.469
C06802=1190.588,311.982,-70.952,-176.559,7.678,148.469
C06803=1190.592,311.734,-70.922,-176.561,7.675,148.469
C06804=1190.597,311.486,-70.891,-176.564,7.672,148.469
C06805=1190.601,311.238,-70.861,-176.566,7.669,148.469
C06806=1190.605,310.990,-70.830,-176.569,7.666,148.469
C06807=1190.610,310.742,-70.799,-176.571,7.664,148.469
C06808=1190.613,310.494,-70.769,-176.573,7.661,148.469
C06809=1190.618,310.246,-70.739,-176.576,7.658,148.469
C06810=1190.622,309.997,-70.708,-176.579,7.655,148.469
C06811=1190.626,309.749,-70.677,-176.581,7.651,148.469
C06812=1190.631,309.501,-70.647,-176.583,7.649,148.469
C06813=1190.635,309.254,-70.616,-176.586,7.646,148.469
C06814=1190.639,309.005,-70.585,-176.589,7.643,148.469
C06815=1190.644,308.756,-70.555,-176.591,7.640,148.469
C06816=1190.648,308.509,-70.525,-176.594,7.637,148.469
C06817=1190.652,308.261,-70.494,-176.596,7.635,148.469
C06818=1190.656,308.013,-70.464,-176.598,7.631,148.469
C06819=1190.660,307.764,-70.433,-176.601,7.628,148.469
C06820=1190.665,307.516,-70.403,-176.604,7.625,148.469
C06821=1190.669,307.268,-70.373,-176.606,7.623,148.469
C06822=1190.673,307.020,-70.342,-176.608,7.620,148.469
C06823=1190.677,306.773,-70.312,-176.611,7.617,148.469
C06824=1190.682,306.523,-70.281,-176.614,7.614,148.469
C06825=1190.686,306.276,-70.251,-176.616,7.611,148.469
C06826=1190.690,306.028,-70.221,-176.618,7.608,148.469
C06827=1190.694,305.779,-70.191,-176.621,7.605,148.469
C06828=1190.699,305.532,-70.160,-176.623,7.602,148.469
C06829=1190.703,305.284,-70.130,-176.626,7.599,148.469
C06830=1190.708,305.035,-70.100,-176.628,7.597,148.469
C06831=1190.711,304.787,-70.070,-176.631,7.594,148.469
C06832=1190.716,304.538,-70.039,-176.634,7.591,148.469
C06833=1190.720,304.291,-70.009,-176.636,7.588,148.469
C06834=1190.724,304.043,-69.979,-176.638,7.586,148.469
C06835=1190.729,303.794,-69.949,-176.641,7.583,148.469
C06836=1190.733,303.547,-69.918,-176.644,7.580,148.469
C06837=1190.737,303.298,-69.889,-176.646,7.577,148.469
C06838=1190.741,303.051,-69.859,-176.649,7.574,148.469
C06839=1190.746,302.802,-69.829,-176.651,7.572,148.469
C06840=1190.749,302.554,-69.798,-176.653,7.568,148.469
C06841=1190.754,302.305,-69.768,-176.656,7.565,148.469
C06842=1190.758,302.057,-69.738,-176.659,7.562,148.469
C06843=1190.762,301.809,-69.708,-176.661,7.560,148.469
C06844=1190.767,301.561,-69.678,-176.664,7.557,148.469
C06845=1190.771,301.313,-69.648,-176.666,7.554,148.469
C06846=1190.775,301.065,-69.619,-176.669,7.551,148.469
C06847=1190.780,300.817,-69.588,-176.671,7.549,148.469
C06848=1190.784,300.568,-69.559,-176.673,7.546,148.469
C06849=1190.788,300.321,-69.528,-176.676,7.543,148.469
C06850=1190.793,300.072,-69.498,-176.679,7.540,148.469
C06851=1190.797,299.824,-69.469,-176.681,7.537,148.469
C06852=1190.801,299.576,-69.439,-176.684,7.534,148.469
C06853=1190.806,299.328,-69.409,-176.686,7.531,148.469
C06854=1190.810,299.080,-69.379,-176.689,7.528,148.469
C06855=1190.814,298.832,-69.349,-176.691,7.526,148.469
C06856=1190.818,298.584,-69.320,-176.694,7.523,148.469
C06857=1190.823,298.335,-69.290,-176.697,7.520,148.469
C06858=1190.827,298.087,-69.260,-176.699,7.518,148.469
C06859=1190.831,297.839,-69.230,-176.702,7.515,148.469
C06860=1190.835,297.591,-69.200,-176.704,7.512,148.469
C06861=1190.840,297.342,-69.170,-176.706,7.509,148.469
C06862=1190.844,297.094,-69.141,-176.709,7.506,148.469
C06863=1190.848,296.846,-69.111,-176.711,7.503,148.469
C06864=1190.853,296.598,-69.081,-176.714,7.500,148.469
C06865=1190.857,296.350,-69.052,-176.717,7.497,148.469
C06866=1190.862,296.101,-69.022,-176.719,7.495,148.469
C06867=1190.866,295.853,-68.992,-176.722,7.492,148.469
C06868=1190.870,295.605,-68.963,-176.724,7.489,148.469
C06869=1190.874,295.357,-68.933,-176.727,7.486,148.469
C06870=1190.878,295.109,-68.903,-176.729,7.484,148.469
C06871=1190.882,294.861,-68.874,-176.732,7.481,148.469
C06872=1190.886,294.612,-68.844,-176.735,7.478,148.469
C06873=1190.891,294.364,-68.814,-176.737,7.476,148.469
C06874=1190.896,294.115,-68.785,-176.739,7.473,148.469
C06875=1190.900,293.867,-68.755,-176.742,7.470,148.469
C06876=1190.904,293.619,-68.726,-176.745,7.467,148.469
C06877=1190.908,293.371,-68.697,-176.747,7.465,148.470
C06878=1190.912,293.122,-68.667,-176.750,7.462,148.470
C06879=1190.916,292.874,-68.638,-176.752,7.459,148.470
C06880=1190.921,292.626,-68.609,-176.755,7.457,148.470
C06881=1190.925,292.378,-68.579,-176.757,7.454,148.470
C06882=1190.930,292.130,-68.550,-176.760,7.451,148.470
C06883=1190.934,291.882,-68.520,-176.762,7.448,148.470
C06884=1190.938,291.633,-68.491,-176.765,7.445,148.470
C06885=1190.942,291.385,-68.461,-176.768,7.442,148.470
C06886=1190.946,291.137,-68.432,-176.770,7.439,148.470
C06887=1190.950,290.889,-68.402,-176.772,7.437,148.470
C06888=1190.955,290.641,-68.373,-176.775,7.434,148.470
C06889=1190.960,290.392,-68.345,-176.778,7.431,148.470
C06890=1190.964,290.144,-68.315,-176.780,7.429,148.470
C06891=1190.968,289.896,-68.286,-176.783,7.426,148.470
C06892=1190.972,289.647,-68.256,-176.785,7.423,148.470
C06893=1190.976,289.399,-68.227,-176.788,7.421,148.470
C06894=1190.981,289.152,-68.198,-176.790,7.418,148.470
C06895=1190.986,288.876,-68.165,-176.793,7.415,148.470
C06896=1190.991,288.602,-68.133,-176.796,7.412,148.470
C06897=1190.995,288.327,-68.101,-176.798,7.409,148.470
C06898=1191.000,288.053,-68.068,-176.801,7.406,148.470
C06899=1191.005,287.804,-68.039,-176.804,7.403,148.470
C06900=1191.009,287.556,-68.010,-176.807,7.400,148.470
C06901=1191.013,287.308,-67.982,-176.809,7.398,148.470
C06902=1191.017,287.060,-67.952,-176.812,7.395,148.471
C06903=1191.022,286.812,-67.923,-176.815,7.392,148.471
C06904=1191.026,286.563,-67.894,-176.817,7.390,148.471
C06905=1191.031,286.315,-67.865,-176.819,7.387,148.471
C06906=1191.035,286.067,-67.836,-176.822,7.384,148.471
C06907=1191.039,285.818,-67.807,-176.825,7.381,148.471
C06908=1191.043,285.570,-67.778,-176.827,7.379,148.471
C06909=1191.048,285.323,-67.749,-176.830,7.376,148.471
C06910=1191.052,285.074,-67.720,-176.832,7.373,148.471
C06911=1191.056,284.825,-67.691,-176.835,7.370,148.471
C06912=1191.061,284.577,-67.662,-176.837,7.367,148.471
C06913=1191.066,284.329,-67.633,-176.839,7.365,148.471
C06914=1191.069,284.080,-67.605,-176.842,7.362,148.471
C06915=1191.074,283.832,-67.575,-176.845,7.359,148.471
C06916=1191.078,283.583,-67.547,-176.847,7.357,148.471
C06917=1191.083,283.336,-67.517,-176.850,7.354,148.472
C06918=1191.087,283.087,-67.489,-176.853,7.351,148.472
C06919=1191.091,282.839,-67.460,-176.855,7.349,148.472
C06920=1191.096,282.591,-67.432,-176.858,7.346,148.472
C06921=1191.100,282.342,-67.402,-176.861,7.343,148.472
C06922=1191.104,282.094,-67.374,-176.863,7.341,148.472
C06923=1191.109,281.846,-67.345,-176.865,7.338,148.472
C06924=1191.113,281.597,-67.316,-176.868,7.335,148.472
C06925=1191.117,281.349,-67.287,-176.870,7.333,148.472
C06926=1191.122,281.101,-67.259,-176.873,7.330,148.472
C06927=1191.126,280.852,-67.230,-176.876,7.327,148.472
C06928=1191.130,280.604,-67.201,-176.878,7.325,148.472
C06929=1191.135,280.356,-67.173,-176.881,7.322,148.472
C06930=1191.139,280.108,-67.143,-176.883,7.320,148.472
C06931=1191.143,279.859,-67.115,-176.886,7.317,148.472
C06932=1191.148,279.611,-67.087,-176.889,7.314,148.472
C06933=1191.152,279.363,-67.057,-176.891,7.312,148.473
C06934=1191.156,279.114,-67.029,-176.893,7.309,148.473
C06935=1191.161,278.866,-67.001,-176.897,7.306,148.473
C06936=1191.165,278.617,-66.972,-176.899,7.304,148.473
C06937=1191.169,278.370,-66.944,-176.902,7.301,148.473
C06938=1191.174,278.121,-66.915,-176.904,7.298,148.473
C06939=1191.177,277.873,-66.887,-176.906,7.296,148.473
C06940=1191.182,277.624,-66.858,-176.909,7.293,148.473
C06941=1191.186,277.376,-66.830,-176.911,7.290,148.473
C06942=1191.190,277.127,-66.801,-176.914,7.287,148.473
C06943=1191.196,276.879,-66.773,-176.917,7.285,148.473
C06944=1191.199,276.631,-66.744,-176.919,7.283,148.474
C06945=1191.204,276.383,-66.716,-176.922,7.280,148.474
C06946=1191.208,276.134,-66.688,-176.924,7.277,148.474
C06947=1191.213,275.886,-66.659,-176.927,7.274,148.474
C06948=1191.217,275.638,-66.631,-176.930,7.271,148.474
C06949=1191.221,275.389,-66.602,-176.932,7.270,148.474
C06950=1191.225,275.141,-66.574,-176.935,7.267,148.474
C06951=1191.230,274.892,-66.545,-176.937,7.264,148.474
C06952=1191.234,274.644,-66.518,-176.940,7.261,148.474
C06953=1191.239,274.395,-66.489,-176.943,7.258,148.474
C06954=1191.243,274.148,-66.461,-176.945,7.256,148.474
C06955=1191.247,273.899,-66.433,-176.948,7.254,148.475
C06956=1191.252,273.651,-66.405,-176.950,7.251,148.475
C06957=1191.256,273.402,-66.376,-176.953,7.248,148.475
C06958=1191.261,273.154,-66.348,-176.955,7.245,148.475
C06959=1191.265,272.905,-66.320,-176.958,7.243,148.475
C06960=1191.270,272.657,-66.292,-176.961,7.241,148.475
C06961=1191.273,272.409,-66.263,-176.963,7.238,148.475
C06962=1191.278,272.161,-66.236,-176.966,7.235,148.475
C06963=1191.282,271.912,-66.207,-176.968,7.232,148.475
C06964=1191.287,271.664,-66.179,-176.971,7.230,148.475
C06965=1191.291,271.415,-66.150,-176.974,7.228,148.476
C06966=1191.295,271.167,-66.123,-176.976,7.225,148.476
C06967=1191.299,270.919,-66.094,-176.979,7.222,148.476
C06968=1191.304,270.671,-66.066,-176.981,7.220,148.476
C06969=1191.308,270.422,-66.038,-176.983,7.217,148.476
C06970=1191.313,270.173,-66.011,-176.987,7.215,148.476
C06971=1191.317,269.925,-65.982,-176.989,7.212,148.476
C06972=1191.322,269.677,-65.954,-176.992,7.209,148.476
C06973=1191.326,269.429,-65.927,-176.994,7.207,148.476
C06974=1191.330,269.180,-65.898,-176.996,7.204,148.476
C06975=1191.335,268.931,-65.871,-176.999,7.202,148.477
C06976=1191.339,268.683,-65.843,-177.002,7.199,148.477
C06977=1191.343,268.435,-65.815,-177.004,7.196,148.477
C06978=1191.348,268.187,-65.786,-177.007,7.194,148.477
C06979=1191.352,267.938,-65.758,-177.010,7.192,148.477
C06980=1191.357,267.690,-65.731,-177.012,7.189,148.477
C06981=1191.360,267.441,-65.703,-177.015,7.186,148.477
C06982=1191.365,267.193,-65.675,-177.017,7.184,148.477
C06983=1191.370,266.944,-65.648,-177.020,7.182,148.478
C06984=1191.374,266.696,-65.620,-177.022,7.179,148.478
C06985=1191.378,266.448,-65.592,-177.025,7.176,148.478
C06986=1191.383,266.198,-65.564,-177.027,7.174,148.478
C06987=1191.387,265.951,-65.536,-177.030,7.172,148.478
C06988=1191.392,265.703,-65.508,-177.033,7.169,148.478
C06989=1191.396,265.454,-65.481,-177.035,7.166,148.478
C06990=1191.400,265.206,-65.453,-177.038,7.163,148.478
C06991=1191.405,264.957,-65.426,-177.040,7.162,148.478
C06992=1191.409,264.708,-65.397,-177.043,7.159,148.479
C06993=1191.414,264.460,-65.369,-177.045,7.156,148.479
C06994=1191.418,264.212,-65.342,-177.048,7.153,148.479
C06995=1191.422,263.963,-65.314,-177.051,7.152,148.479
C06996=1191.427,263.715,-65.287,-177.053,7.149,148.479
C06997=1191.431,263.467,-65.259,-177.056,7.146,148.479
C06998=1191.435,263.218,-65.232,-177.059,7.144,148.479
C06999=1191.440,262.945,-65.202,-177.061,7.141,148.479
C07000=1191.446,262.673,-65.171,-177.064,7.138,148.479
C07001=1191.450,262.399,-65.141,-177.067,7.136,148.480
C07002=1191.455,262.127,-65.111,-177.070,7.133,148.480
C07003=1191.459,261.878,-65.083,-177.073,7.130,148.480
C07004=1191.463,261.630,-65.056,-177.075,7.128,148.480
C07005=1191.468,261.381,-65.029,-177.078,7.125,148.480
C07006=1191.473,261.133,-65.000,-177.080,7.123,148.480
C07007=1191.477,260.884,-64.973,-177.083,7.120,148.481
C07008=1191.481,260.636,-64.945,-177.085,7.118,148.481
C07009=1191.486,260.388,-64.918,-177.088,7.115,148.481
C07010=1191.490,260.138,-64.891,-177.090,7.113,148.481
C07011=1191.494,259.890,-64.863,-177.093,7.110,148.481
C07012=1191.499,259.642,-64.836,-177.095,7.108,148.481
C07013=1191.504,259.393,-64.809,-177.099,7.105,148.481
C07014=1191.508,259.146,-64.781,-177.101,7.103,148.482
C07015=1191.511,258.897,-64.754,-177.103,7.100,148.482
C07016=1191.516,258.648,-64.727,-177.106,7.098,148.482
C07017=1191.521,258.400,-64.700,-177.109,7.095,148.482
C07018=1191.525,258.152,-64.672,-177.111,7.093,148.482
C07019=1191.529,257.903,-64.645,-177.114,7.091,148.482
C07020=1191.534,257.654,-64.618,-177.116,7.088,148.482
C07021=1191.538,257.406,-64.591,-177.119,7.085,148.482
C07022=1191.543,257.158,-64.563,-177.122,7.084,148.483
C07023=1191.547,256.909,-64.536,-177.124,7.081,148.483
C07024=1191.551,256.660,-64.508,-177.127,7.078,148.483
C07025=1191.556,256.412,-64.481,-177.130,7.076,148.483
C07026=1191.561,256.163,-64.454,-177.132,7.074,148.483
C07027=1191.565,255.915,-64.428,-177.135,7.071,148.483
C07028=1191.569,255.667,-64.400,-177.137,7.069,148.484
C07029=1191.574,255.419,-64.373,-177.140,7.066,148.484
C07030=1191.578,255.169,-64.346,-177.142,7.064,148.484
C07031=1191.582,254.921,-64.318,-177.145,7.062,148.484
C07032=1191.587,254.672,-64.291,-177.147,7.059,148.484
C07033=1191.592,254.424,-64.264,-177.150,7.057,148.484
C07034=1191.596,254.176,-64.238,-177.153,7.054,148.484
C07035=1191.600,253.927,-64.211,-177.155,7.052,148.485
C07036=1191.605,253.679,-64.184,-177.158,7.049,148.485
C07037=1191.609,253.429,-64.156,-177.160,7.047,148.485
C07038=1191.614,253.181,-64.129,-177.163,7.044,148.485
C07039=1191.618,252.933,-64.103,-177.166,7.042,148.485
C07040=1191.622,252.684,-64.076,-177.168,7.039,148.485
C07041=1191.627,252.436,-64.049,-177.171,7.037,148.486
C07042=1191.632,252.187,-64.022,-177.173,7.035,148.486
C07043=1191.636,251.939,-63.995,-177.176,7.032,148.486
C07044=1191.640,251.691,-63.968,-177.179,7.030,148.486
C07045=1191.645,251.442,-63.941,-177.181,7.027,148.486
C07046=1191.649,251.194,-63.914,-177.183,7.025,148.486
C07047=1191.653,250.945,-63.887,-177.187,7.023,148.487
C07048=1191.657,250.696,-63.860,-177.189,7.020,148.487
C07049=1191.662,250.448,-63.833,-177.191,7.019,148.487
C07050=1191.666,250.200,-63.807,-177.194,7.016,148.487
C07051=1191.671,249.950,-63.780,-177.197,7.014,148.487
C07052=1191.676,249.702,-63.753,-177.200,7.011,148.487
C07053=1191.680,249.454,-63.727,-177.202,7.009,148.487
C07054=1191.684,249.205,-63.700,-177.205,7.006,148.488
C07055=1191.689,248.957,-63.673,-177.207,7.004,148.488
C07056=1191.693,248.709,-63.646,-177.210,7.002,148.488
C07057=1191.698,248.460,-63.620,-177.212,6.999,148.488
C07058=1191.702,248.211,-63.593,-177.215,6.997,148.488
C07059=1191.706,247.963,-63.566,-177.218,6.994,148.489
C07060=1191.711,247.714,-63.539,-177.220,6.992,148.489
C07061=1191.715,247.466,-63.513,-177.223,6.990,148.489
C07062=1191.720,247.217,-63.486,-177.225,6.987,148.489
C07063=1191.725,246.969,-63.459,-177.228,6.985,148.489
C07064=1191.728,246.720,-63.433,-177.231,6.982,148.489
C07065=1191.733,246.471,-63.406,-177.233,6.980,148.490
C07066=1191.737,246.223,-63.380,-177.236,6.977,148.490
C07067=1191.742,245.975,-63.353,-177.238,6.975,148.490
C07068=1191.746,245.726,-63.327,-177.241,6.973,148.490
C07069=1191.751,245.477,-63.300,-177.244,6.970,148.490
C07070=1191.755,245.228,-63.274,-177.246,6.969,148.491
C07071=1191.760,244.980,-63.247,-177.248,6.966,148.491
C07072=1191.764,244.732,-63.221,-177.252,6.964,148.491
C07073=1191.769,244.483,-63.194,-177.254,6.962,148.491
C07074=1191.773,244.234,-63.168,-177.257,6.959,148.491
C07075=1191.778,243.985,-63.142,-177.259,6.957,148.491
C07076=1191.781,243.737,-63.115,-177.262,6.955,148.492
C07077=1191.787,243.489,-63.089,-177.264,6.952,148.492
C07078=1191.791,243.241,-63.063,-177.267,6.950,148.492
C07079=1191.796,242.992,-63.036,-177.270,6.947,148.492
C07080=1191.800,242.743,-63.010,-177.272,6.945,148.492
C07081=1191.804,242.495,-62.983,-177.275,6.943,148.493
C07082=1191.809,242.246,-62.957,-177.277,6.940,148.493
C07083=1191.813,241.997,-62.930,-177.280,6.938,148.493
C07084=1191.818,241.749,-62.904,-177.282,6.936,148.493
C07085=1191.821,241.500,-62.878,-177.285,6.934,148.493
C07086=1191.826,241.251,-62.852,-177.288,6.931,148.493
C07087=1191.831,241.003,-62.826,-177.291,6.929,148.494
C07088=1191.836,240.755,-62.799,-177.293,6.927,148.494
C07089=1191.840,240.506,-62.773,-177.296,6.925,148.494
C07090=1191.844,240.258,-62.747,-177.298,6.922,148.494
C07091=1191.849,240.009,-62.721,-177.301,6.920,148.495
C07092=1191.853,239.760,-62.695,-177.303,6.918,148.495
C07093=1191.857,239.512,-62.668,-177.306,6.915,148.495
C07094=1191.862,239.263,-62.642,-177.308,6.913,148.495
C07095=1191.867,239.014,-62.617,-177.311,6.911,148.495
C07096=1191.871,238.766,-62.590,-177.314,6.908,148.495
C07097=1191.876,238.517,-62.564,-177.316,6.906,148.496
C07098=1191.880,238.268,-62.538,-177.319,6.905,148.496
C07099=1191.884,238.020,-62.512,-177.322,6.902,148.496
C07100=1191.889,237.771,-62.485,-177.324,6.900,148.496
C07101=1191.894,237.523,-62.460,-177.327,6.898,148.497
C07102=1191.898,237.274,-62.434,-177.330,6.895,148.497
C07103=1191.902,237.003,-62.405,-177.332,6.893,148.497
C07104=1191.908,236.731,-62.377,-177.335,6.890,148.497
C07105=1191.913,236.460,-62.348,-177.338,6.887,148.497
C07106=1191.917,236.188,-62.320,-177.341,6.885,148.498
C07107=1191.922,235.939,-62.294,-177.344,6.883,148.498
C07108=1191.927,235.690,-62.268,-177.346,6.880,148.498
C07109=1191.931,235.443,-62.242,-177.349,6.879,148.498
C07110=1191.935,235.194,-62.216,-177.352,6.876,148.499
C07111=1191.940,234.945,-62.191,-177.354,6.874,148.499
C07112=1191.944,234.696,-62.165,-177.357,6.872,148.499
C07113=1191.949,234.448,-62.139,-177.359,6.869,148.499
C07114=1191.954,234.199,-62.113,-177.362,6.867,148.499
C07115=1191.958,233.950,-62.087,-177.364,6.865,148.500
C07116=1191.962,233.702,-62.062,-177.367,6.862,148.500
C07117=1191.967,233.454,-62.035,-177.370,6.861,148.500
C07118=1191.971,233.205,-62.010,-177.372,6.858,148.500
C07119=1191.976,232.956,-61.983,-177.375,6.856,148.501
C07120=1191.980,232.707,-61.958,-177.377,6.854,148.501
C07121=1191.985,232.459,-61.932,-177.380,6.852,148.501
C07122=1191.989,232.210,-61.906,-177.382,6.850,148.501
C07123=1191.993,231.962,-61.881,-177.385,6.847,148.501
C07124=1191.998,231.714,-61.855,-177.388,6.845,148.502
C07125=1192.002,231.465,-61.830,-177.390,6.843,148.502
C07126=1192.007,231.216,-61.804,-177.394,6.840,148.502
C07127=1192.011,230.968,-61.778,-177.396,6.838,148.502
C07128=1192.017,230.718,-61.753,-177.398,6.836,148.503
C07129=1192.021,230.469,-61.727,-177.402,6.834,148.503
C07130=1192.025,230.220,-61.701,-177.404,6.832,148.503
C07131=1192.030,229.972,-61.676,-177.406,6.830,148.503
C07132=1192.034,229.724,-61.650,-177.409,6.828,148.503
C07133=1192.038,229.475,-61.624,-177.412,6.825,148.504
C07134=1192.043,229.227,-61.599,-177.414,6.823,148.504
C07135=1192.047,228.978,-61.573,-177.417,6.821,148.504
C07136=1192.052,228.730,-61.548,-177.420,6.818,148.504
C07137=1192.057,228.480,-61.523,-177.422,6.816,148.504
C07138=1192.061,228.231,-61.497,-177.425,6.814,148.505
C07139=1192.066,227.983,-61.472,-177.427,6.812,148.505
C07140=1192.070,227.735,-61.446,-177.430,6.809,148.505
C07141=1192.074,227.486,-61.420,-177.433,6.808,148.506
C07142=1192.079,227.237,-61.396,-177.435,6.806,148.506
C07143=1192.084,226.988,-61.370,-177.437,6.804,148.506
C07144=1192.089,226.740,-61.344,-177.441,6.801,148.506
C07145=1192.093,226.491,-61.319,-177.443,6.799,148.507
C07146=1192.097,226.242,-61.294,-177.445,6.797,148.507
C07147=1192.101,225.994,-61.269,-177.449,6.794,148.507
C07148=1192.106,225.745,-61.243,-177.451,6.792,148.507
C07149=1192.111,225.497,-61.218,-177.453,6.790,148.507
C07150=1192.115,225.248,-61.193,-177.456,6.789,148.508
C07151=1192.119,224.999,-61.167,-177.459,6.786,148.508
C07152=1192.124,224.750,-61.142,-177.461,6.784,148.508
C07153=1192.129,224.501,-61.117,-177.464,6.782,148.508
C07154=1192.133,224.253,-61.091,-177.466,6.780,148.509
C07155=1192.138,224.004,-61.066,-177.469,6.777,148.509
C07156=1192.142,223.756,-61.041,-177.472,6.775,148.509
C07157=1192.146,223.507,-61.016,-177.474,6.773,148.509
C07158=1192.151,223.259,-60.991,-177.477,6.771,148.510
C07159=1192.156,223.010,-60.965,-177.480,6.769,148.510
C07160=1192.161,222.761,-60.940,-177.482,6.767,148.510
C07161=1192.165,222.512,-60.915,-177.485,6.765,148.510
C07162=1192.169,222.263,-60.890,-177.488,6.763,148.511
C07163=1192.174,222.015,-60.865,-177.490,6.760,148.511
C07164=1192.178,221.766,-60.840,-177.493,6.758,148.511
C07165=1192.183,221.518,-60.814,-177.496,6.756,148.511
C07166=1192.187,221.268,-60.789,-177.498,6.754,148.512
C07167=1192.191,221.020,-60.765,-177.501,6.752,148.512
C07168=1192.196,220.771,-60.740,-177.504,6.750,148.512
C07169=1192.201,220.523,-60.714,-177.506,6.748,148.513
C07170=1192.205,220.273,-60.689,-177.509,6.746,148.513
C07171=1192.209,220.026,-60.664,-177.511,6.744,148.513
C07172=1192.215,219.777,-60.640,-177.514,6.741,148.513
C07173=1192.219,219.528,-60.614,-177.517,6.739,148.513
C07174=1192.224,219.279,-60.589,-177.519,6.737,148.514
C07175=1192.228,219.030,-60.565,-177.522,6.735,148.514
C07176=1192.233,218.782,-60.539,-177.525,6.733,148.514
C07177=1192.237,218.533,-60.514,-177.527,6.731,148.514
C07178=1192.241,218.285,-60.490,-177.530,6.729,148.515
C07179=1192.246,218.035,-60.465,-177.533,6.727,148.515
C07180=1192.251,217.787,-60.440,-177.535,6.724,148.515
C07181=1192.254,217.538,-60.415,-177.538,6.722,148.516
C07182=1192.259,217.290,-60.390,-177.541,6.720,148.516
C07183=1192.265,217.041,-60.365,-177.543,6.718,148.516
C07184=1192.268,216.792,-60.341,-177.545,6.716,148.516
C07185=1192.273,216.544,-60.316,-177.549,6.714,148.517
C07186=1192.277,216.294,-60.291,-177.551,6.712,148.517
C07187=1192.282,216.046,-60.267,-177.553,6.710,148.517
C07188=1192.287,215.797,-60.242,-177.556,6.708,148.517
C07189=1192.291,215.549,-60.217,-177.559,6.706,148.518
C07190=1192.296,215.300,-60.192,-177.562,6.704,148.518
C07191=1192.300,215.051,-60.168,-177.564,6.701,148.518
C07192=1192.305,214.802,-60.143,-177.567,6.700,148.519
C07193=1192.310,214.553,-60.118,-177.569,6.698,148.519
C07194=1192.313,214.305,-60.093,-177.572,6.696,148.519
C07195=1192.319,214.056,-60.068,-177.575,6.693,148.519
C07196=1192.323,213.808,-60.044,-177.577,6.691,148.520
C07197=1192.327,213.558,-60.019,-177.580,6.689,148.520
C07198=1192.332,213.310,-59.995,-177.583,6.688,148.520
C07199=1192.337,213.061,-59.971,-177.585,6.685,148.520
C07200=1192.341,212.812,-59.946,-177.588,6.683,148.521
C07201=1192.346,212.563,-59.921,-177.591,6.681,148.521
C07202=1192.350,212.315,-59.897,-177.593,6.679,148.521
C07203=1192.355,212.066,-59.872,-177.596,6.677,148.521
C07204=1192.359,211.818,-59.848,-177.598,6.675,148.522
C07205=1192.364,211.569,-59.823,-177.601,6.673,148.522
C07206=1192.368,211.320,-59.798,-177.604,6.671,148.522
C07207=1192.373,211.050,-59.772,-177.607,6.669,148.523
C07208=1192.378,210.779,-59.746,-177.610,6.666,148.523
C07209=1192.383,210.508,-59.719,-177.612,6.664,148.523
C07210=1192.388,210.238,-59.692,-177.615,6.662,148.524
C07211=1192.393,209.989,-59.668,-177.618,6.660,148.524
C07212=1192.398,209.741,-59.643,-177.621,6.658,148.524
C07213=1192.402,209.491,-59.619,-177.623,6.656,148.525
C07214=1192.406,209.243,-59.595,-177.626,6.654,148.525
C07215=1192.411,208.994,-59.570,-177.628,6.652,148.525
C07216=1192.415,208.746,-59.546,-177.631,6.649,148.525
C07217=1192.420,208.497,-59.521,-177.634,6.648,148.526
C07218=1192.425,208.247,-59.498,-177.637,6.646,148.526
C07219=1192.429,207.999,-59.473,-177.639,6.644,148.526
C07220=1192.434,207.750,-59.449,-177.642,6.642,148.526
C07221=1192.438,207.501,-59.424,-177.644,6.640,148.527
C07222=1192.442,207.253,-59.400,-177.647,6.637,148.527
C07223=1192.448,207.004,-59.376,-177.650,6.636,148.527
C07224=1192.452,206.756,-59.352,-177.652,6.633,148.528
C07225=1192.457,206.507,-59.328,-177.655,6.632,148.528
C07226=1192.461,206.257,-59.303,-177.658,6.630,148.528
C07227=1192.466,206.009,-59.279,-177.660,6.628,148.529
C07228=1192.470,205.760,-59.255,-177.663,6.626,148.529
C07229=1192.475,205.511,-59.231,-177.666,6.623,148.529
C07230=1192.480,205.263,-59.207,-177.668,6.621,148.529
C07231=1192.484,205.014,-59.183,-177.671,6.620,148.530
C07232=1192.489,204.765,-59.158,-177.674,6.618,148.530
C07233=1192.493,204.516,-59.135,-177.676,6.616,148.530
C07234=1192.498,204.267,-59.110,-177.679,6.614,148.531
C07235=1192.502,204.019,-59.086,-177.681,6.612,148.531
C07236=1192.507,203.769,-59.062,-177.684,6.610,148.531
C07237=1192.511,203.520,-59.038,-177.687,6.608,148.532
C07238=1192.516,203.272,-59.014,-177.690,6.606,148.532
C07239=1192.520,203.023,-58.991,-177.692,6.604,148.532
C07240=1192.525,202.775,-58.966,-177.695,6.602,148.533
C07241=1192.530,202.526,-58.942,-177.697,6.600,148.533
C07242=1192.535,202.277,-58.918,-177.700,6.598,148.533
C07243=1192.539,202.028,-58.894,-177.702,6.596,148.533
C07244=1192.543,201.779,-58.870,-177.705,6.595,148.534
C07245=1192.548,201.530,-58.847,-177.708,6.592,148.534
C07246=1192.552,201.282,-58.822,-177.711,6.590,148.534
C07247=1192.557,201.033,-58.799,-177.713,6.588,148.534
C07248=1192.562,200.784,-58.774,-177.716,6.586,148.535
C07249=1192.567,200.535,-58.751,-177.718,6.584,148.535
C07250=1192.571,200.287,-58.727,-177.721,6.583,148.536
C07251=1192.575,200.037,-58.703,-177.724,6.581,148.536
C07252=1192.579,199.789,-58.679,-177.726,6.579,148.536
C07253=1192.584,199.540,-58.656,-177.729,6.577,148.536
C07254=1192.589,199.291,-58.632,-177.731,6.575,148.537
C07255=1192.594,199.042,-58.608,-177.734,6.572,148.537
C07256=1192.598,198.793,-58.584,-177.737,6.571,148.537
C07257=1192.603,198.544,-58.560,-177.740,6.569,148.538
C07258=1192.607,198.296,-58.536,-177.742,6.567,148.538
C07259=1192.612,198.047,-58.513,-177.745,6.565,148.538
C07260=1192.617,197.798,-58.489,-177.747,6.563,148.538
C07261=1192.621,197.549,-58.466,-177.750,6.561,148.539
C07262=1192.626,197.300,-58.442,-177.753,6.559,148.539
C07263=1192.630,197.052,-58.418,-177.755,6.558,148.540
C07264=1192.635,196.803,-58.395,-177.758,6.556,148.540
C07265=1192.640,196.554,-58.371,-177.761,6.554,148.540
C07266=1192.644,196.306,-58.347,-177.764,6.551,148.541
C07267=1192.649,196.056,-58.324,-177.766,6.550,148.541
C07268=1192.654,195.807,-58.301,-177.769,6.547,148.541
C07269=1192.658,195.559,-58.277,-177.771,6.546,148.541
C07270=1192.663,195.310,-58.253,-177.774,6.544,148.542
C07271=1192.667,195.061,-58.230,-177.777,6.542,148.542
C07272=1192.672,194.813,-58.206,-177.779,6.540,148.542
C07273=1192.676,194.564,-58.182,-177.782,6.538,148.543
C07274=1192.681,194.315,-58.159,-177.785,6.537,148.543
C07275=1192.686,194.065,-58.136,-177.787,6.535,148.543
C07276=1192.690,193.817,-58.112,-177.790,6.533,148.544
C07277=1192.695,193.568,-58.088,-177.792,6.531,148.544
C07278=1192.700,193.319,-58.065,-177.795,6.529,148.544
C07279=1192.704,193.070,-58.041,-177.797,6.527,148.545
C07280=1192.709,192.821,-58.018,-177.800,6.525,148.545
C07281=1192.713,192.573,-57.995,-177.803,6.524,148.545
C07282=1192.717,192.324,-57.971,-177.806,6.521,148.546
C07283=1192.722,192.075,-57.948,-177.809,6.519,148.546
C07284=1192.727,191.826,-57.925,-177.811,6.517,148.546
C07285=1192.731,191.577,-57.901,-177.814,6.516,148.547
C07286=1192.736,191.328,-57.878,-177.817,6.514,148.547
C07287=1192.741,191.079,-57.855,-177.819,6.512,148.547
C07288=1192.746,190.830,-57.831,-177.821,6.510,148.548
C07289=1192.749,190.582,-57.808,-177.824,6.508,148.548
C07290=1192.754,190.332,-57.784,-177.827,6.506,148.548
C07291=1192.759,190.084,-57.761,-177.829,6.504,148.549
C07292=1192.764,189.835,-57.738,-177.832,6.503,148.549
C07293=1192.769,189.586,-57.715,-177.835,6.501,148.549
C07294=1192.773,189.337,-57.691,-177.837,6.499,148.550
C07295=1192.777,189.088,-57.668,-177.840,6.497,148.550
C07296=1192.782,188.839,-57.645,-177.843,6.495,148.550
C07297=1192.787,188.590,-57.622,-177.845,6.494,148.551
C07298=1192.791,188.341,-57.598,-177.848,6.492,148.551
C07299=1192.795,188.092,-57.576,-177.851,6.490,148.551
C07300=1192.801,187.844,-57.553,-177.853,6.488,148.552
C07301=1192.805,187.595,-57.529,-177.856,6.486,148.552
C07302=1192.810,187.346,-57.506,-177.858,6.484,148.552
C07303=1192.814,187.097,-57.483,-177.861,6.483,148.553
C07304=1192.819,186.848,-57.460,-177.864,6.481,148.553
C07305=1192.824,186.599,-57.437,-177.866,6.479,148.553
